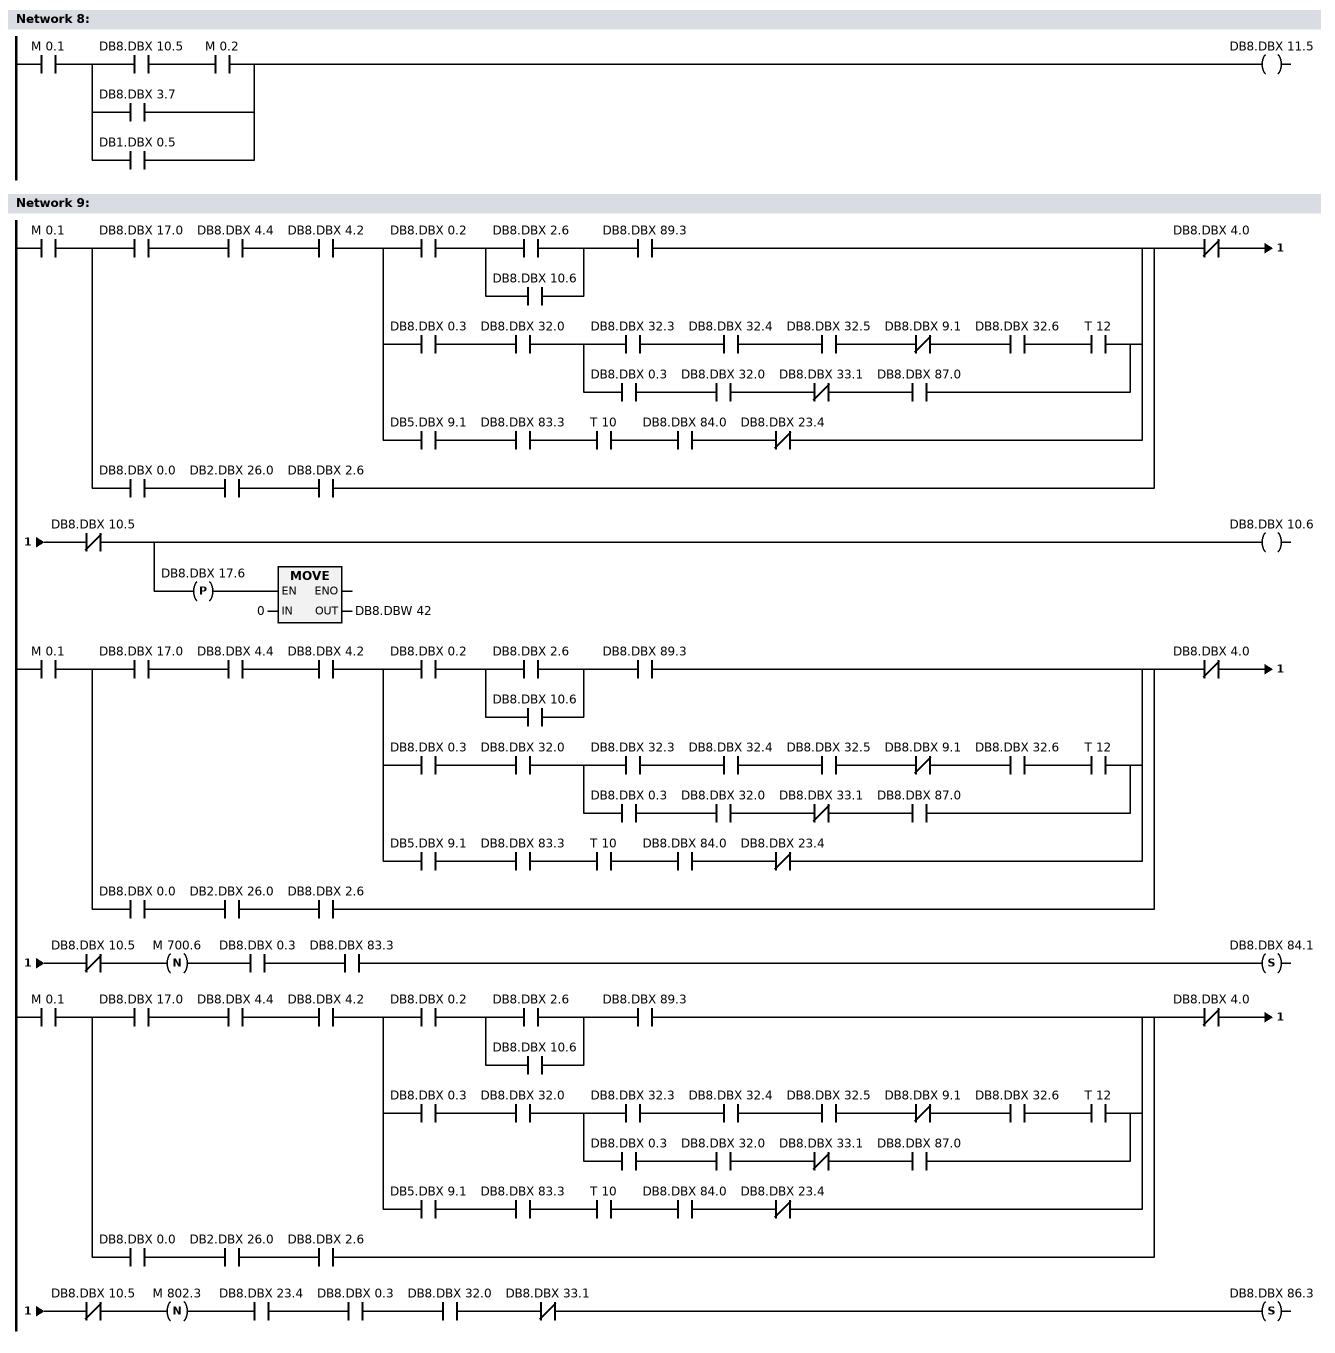
NETWORK
TITLE =
      A     M 0.1;
      A(;
      A     DB8.DBX 10.5;
      A     M 0.2;
      O     DB8.DBX 3.7;
      O     DB1.DBX 0.5;
      );
      =     DB8.DBX 11.5;
NETWORK
TITLE =
      A     M 0.1;
      A(;
      A     DB8.DBX 17.0;
      A     DB8.DBX 4.4;
      A     DB8.DBX 4.2;
      A(;
      A     DB8.DBX 0.2;
      A(;
      O     DB8.DBX 2.6;
      O     DB8.DBX 10.6;
      );
      A     DB8.DBX 89.3;
      O;
      A     DB8.DBX 0.3;
      A     DB8.DBX 32.0;
      A(;
      A     DB8.DBX 32.3;
      A     DB8.DBX 32.4;
      A     DB8.DBX 32.5;
      AN    DB8.DBX 9.1;
      A     DB8.DBX 32.6;
      A     T 12;
      O;
      A     DB8.DBX 0.3;
      A     DB8.DBX 32.0;
      AN    DB8.DBX 33.1;
      A     DB8.DBX 87.0;
      );
      O;
      A     DB5.DBX 9.1;
      A     DB8.DBX 83.3;
      A     T 10;
      A     DB8.DBX 84.0;
      AN    DB8.DBX 23.4;
      );
      O;
      A     DB8.DBX 0.0;
      A     DB2.DBX 26.0;
      A     DB8.DBX 2.6;
      );
      AN    DB8.DBX 4.0;
      AN    DB8.DBX 10.5;
      =     L 0.0;
      A     L 0.0;
      BLD   102;
      =     DB8.DBX 10.6;
      A     L 0.0;
      FP    DB8.DBX 17.6;
      JNB   M003;
      L     0;
      T     DB8.DBW 42;
M003: NOP   0;
      A(;
      A     L 0.0;
      FN    M 700.6;
      );
      A     DB8.DBX 0.3;
      A     DB8.DBX 83.3;
      S     DB8.DBX 84.1;
      A(;
      A     L 0.0;
      FN    M 802.3;
      );
      A     DB8.DBX 23.4;
      A     DB8.DBX 0.3;
      A     DB8.DBX 32.0;
      AN    DB8.DBX 33.1;
      S     DB8.DBX 86.3;
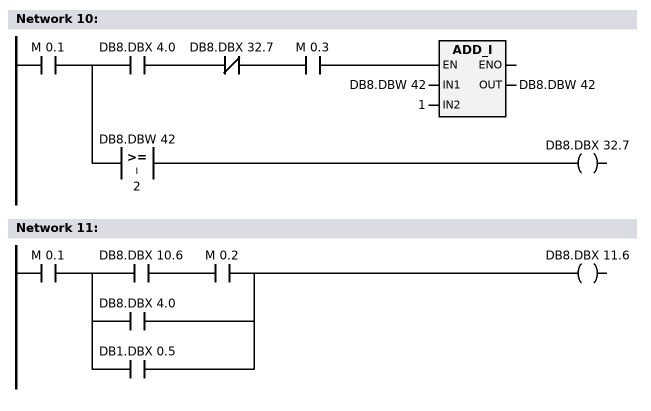
NETWORK
TITLE =
      A     M 0.1;
      =     L 0.0;
      A     L 0.0;
      A     DB8.DBX 4.0;
      AN    DB8.DBX 32.7;
      A     M 0.3;
      JNB   M004;
      L     DB8.DBW 42;
      L     1;
      +I;
      T     DB8.DBW 42;
M004: NOP   0;
      A     L 0.0;
      A(;
      L     DB8.DBW 42;
      L     2;
      >=I;
      );
      =     DB8.DBX 32.7;
NETWORK
TITLE =
      A     M 0.1;
      A(;
      A     DB8.DBX 10.6;
      A     M 0.2;
      O     DB8.DBX 4.0;
      O     DB1.DBX 0.5;
      );
      =     DB8.DBX 11.6;
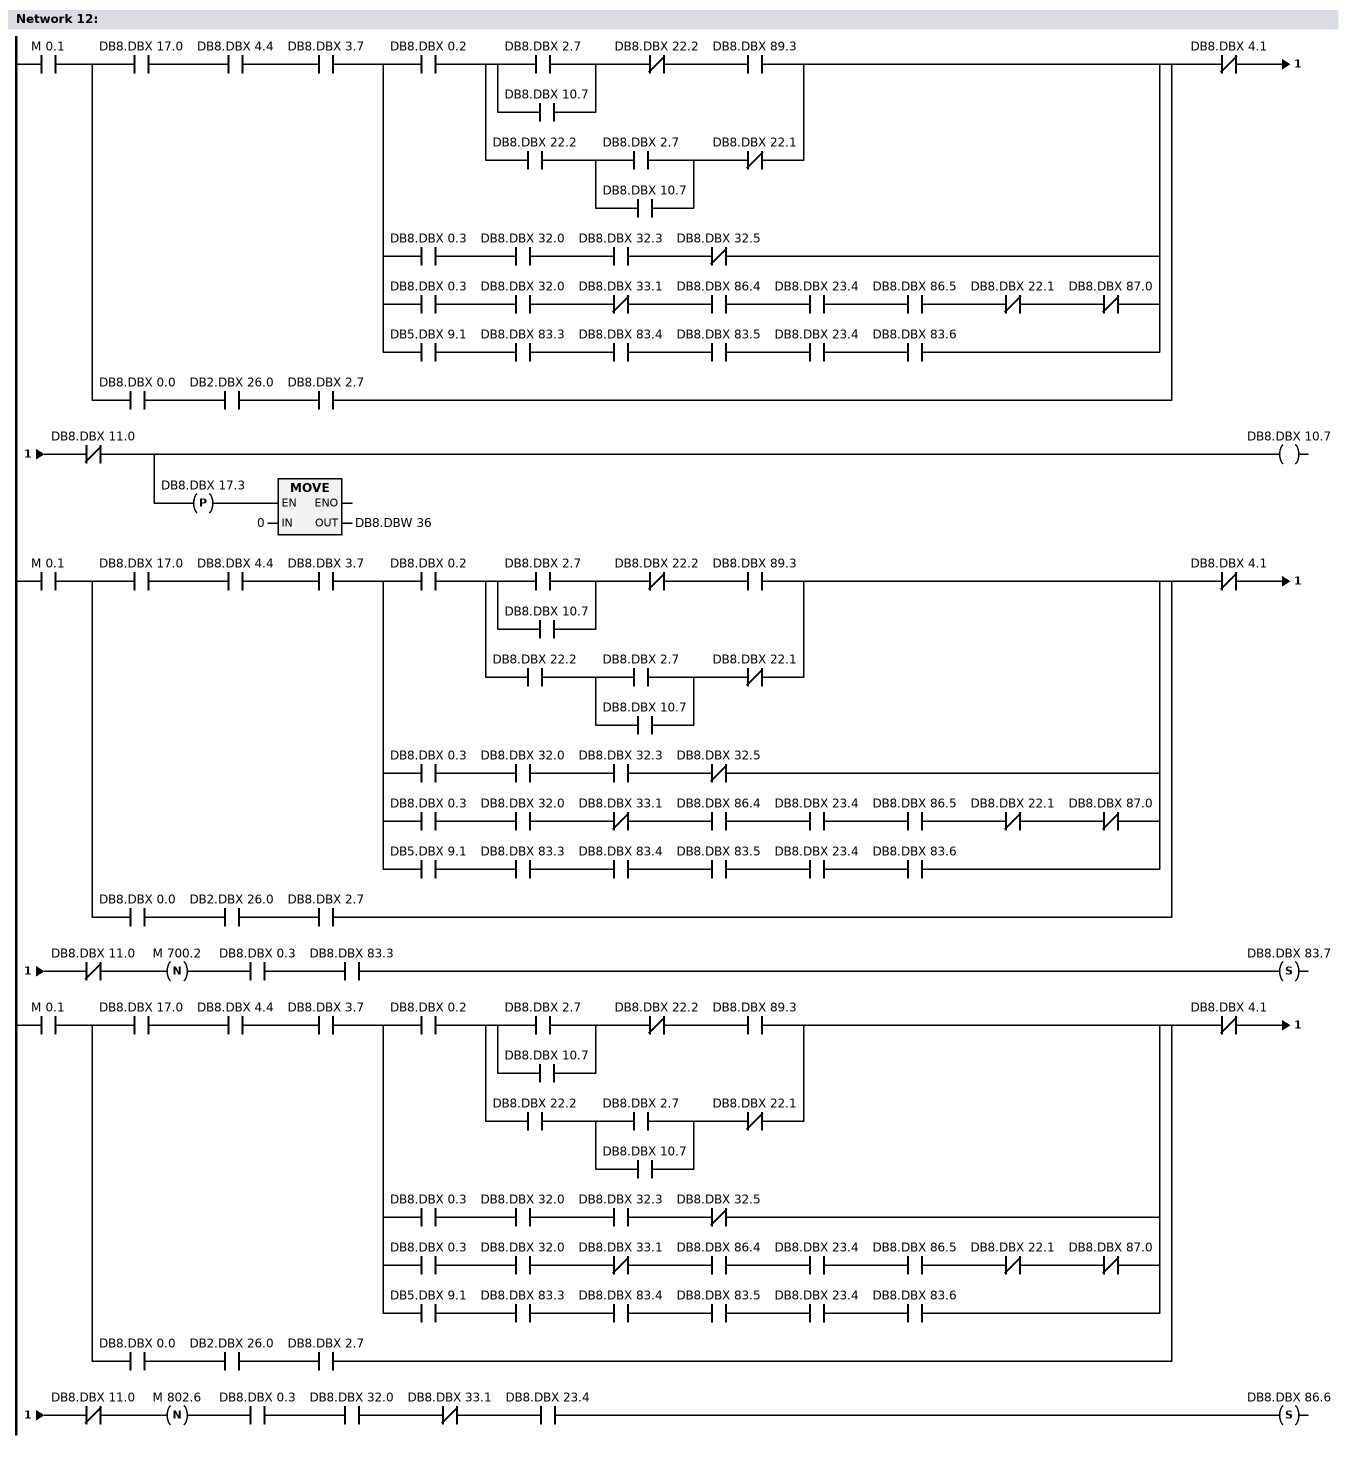
NETWORK
TITLE =
      A     M 0.1;
      A(;
      A     DB8.DBX 17.0;
      A     DB8.DBX 4.4;
      A     DB8.DBX 3.7;
      A(;
      A     DB8.DBX 0.2;
      A(;
      A(;
      O     DB8.DBX 2.7;
      O     DB8.DBX 10.7;
      );
      AN    DB8.DBX 22.2;
      A     DB8.DBX 89.3;
      O;
      A     DB8.DBX 22.2;
      A(;
      O     DB8.DBX 2.7;
      O     DB8.DBX 10.7;
      );
      AN    DB8.DBX 22.1;
      );
      O;
      A     DB8.DBX 0.3;
      A     DB8.DBX 32.0;
      A     DB8.DBX 32.3;
      AN    DB8.DBX 32.5;
      O;
      A     DB8.DBX 0.3;
      A     DB8.DBX 32.0;
      AN    DB8.DBX 33.1;
      A     DB8.DBX 86.4;
      A     DB8.DBX 23.4;
      A     DB8.DBX 86.5;
      AN    DB8.DBX 22.1;
      AN    DB8.DBX 87.0;
      O;
      A     DB5.DBX 9.1;
      A     DB8.DBX 83.3;
      A     DB8.DBX 83.4;
      A     DB8.DBX 83.5;
      A     DB8.DBX 23.4;
      A     DB8.DBX 83.6;
      );
      O;
      A     DB8.DBX 0.0;
      A     DB2.DBX 26.0;
      A     DB8.DBX 2.7;
      );
      AN    DB8.DBX 4.1;
      AN    DB8.DBX 11.0;
      =     L 0.0;
      A     L 0.0;
      BLD   102;
      =     DB8.DBX 10.7;
      A     L 0.0;
      FP    DB8.DBX 17.3;
      JNB   M005;
      L     0;
      T     DB8.DBW 36;
M005: NOP   0;
      A(;
      A     L 0.0;
      FN    M 700.2;
      );
      A     DB8.DBX 0.3;
      A     DB8.DBX 83.3;
      S     DB8.DBX 83.7;
      A(;
      A     L 0.0;
      FN    M 802.6;
      );
      A     DB8.DBX 0.3;
      A     DB8.DBX 32.0;
      AN    DB8.DBX 33.1;
      A     DB8.DBX 23.4;
      S     DB8.DBX 86.6;
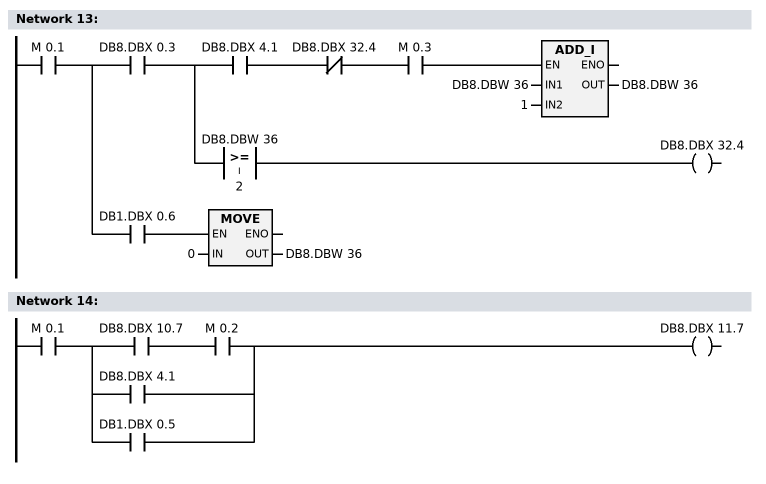
NETWORK
TITLE =
      A     M 0.1;
      =     L 0.0;
      A     L 0.0;
      A     DB8.DBX 0.3;
      =     L 0.1;
      A     L 0.1;
      A     DB8.DBX 4.1;
      AN    DB8.DBX 32.4;
      A     M 0.3;
      JNB   M006;
      L     DB8.DBW 36;
      L     1;
      +I;
      T     DB8.DBW 36;
M006: NOP   0;
      A     L 0.1;
      A(;
      L     DB8.DBW 36;
      L     2;
      >=I;
      );
      =     DB8.DBX 32.4;
      A     L 0.0;
      A     DB1.DBX 0.6;
      JNB   M007;
      L     0;
      T     DB8.DBW 36;
M007: NOP   0;
NETWORK
TITLE =
      A     M 0.1;
      A(;
      A     DB8.DBX 10.7;
      A     M 0.2;
      O     DB8.DBX 4.1;
      O     DB1.DBX 0.5;
      );
      =     DB8.DBX 11.7;
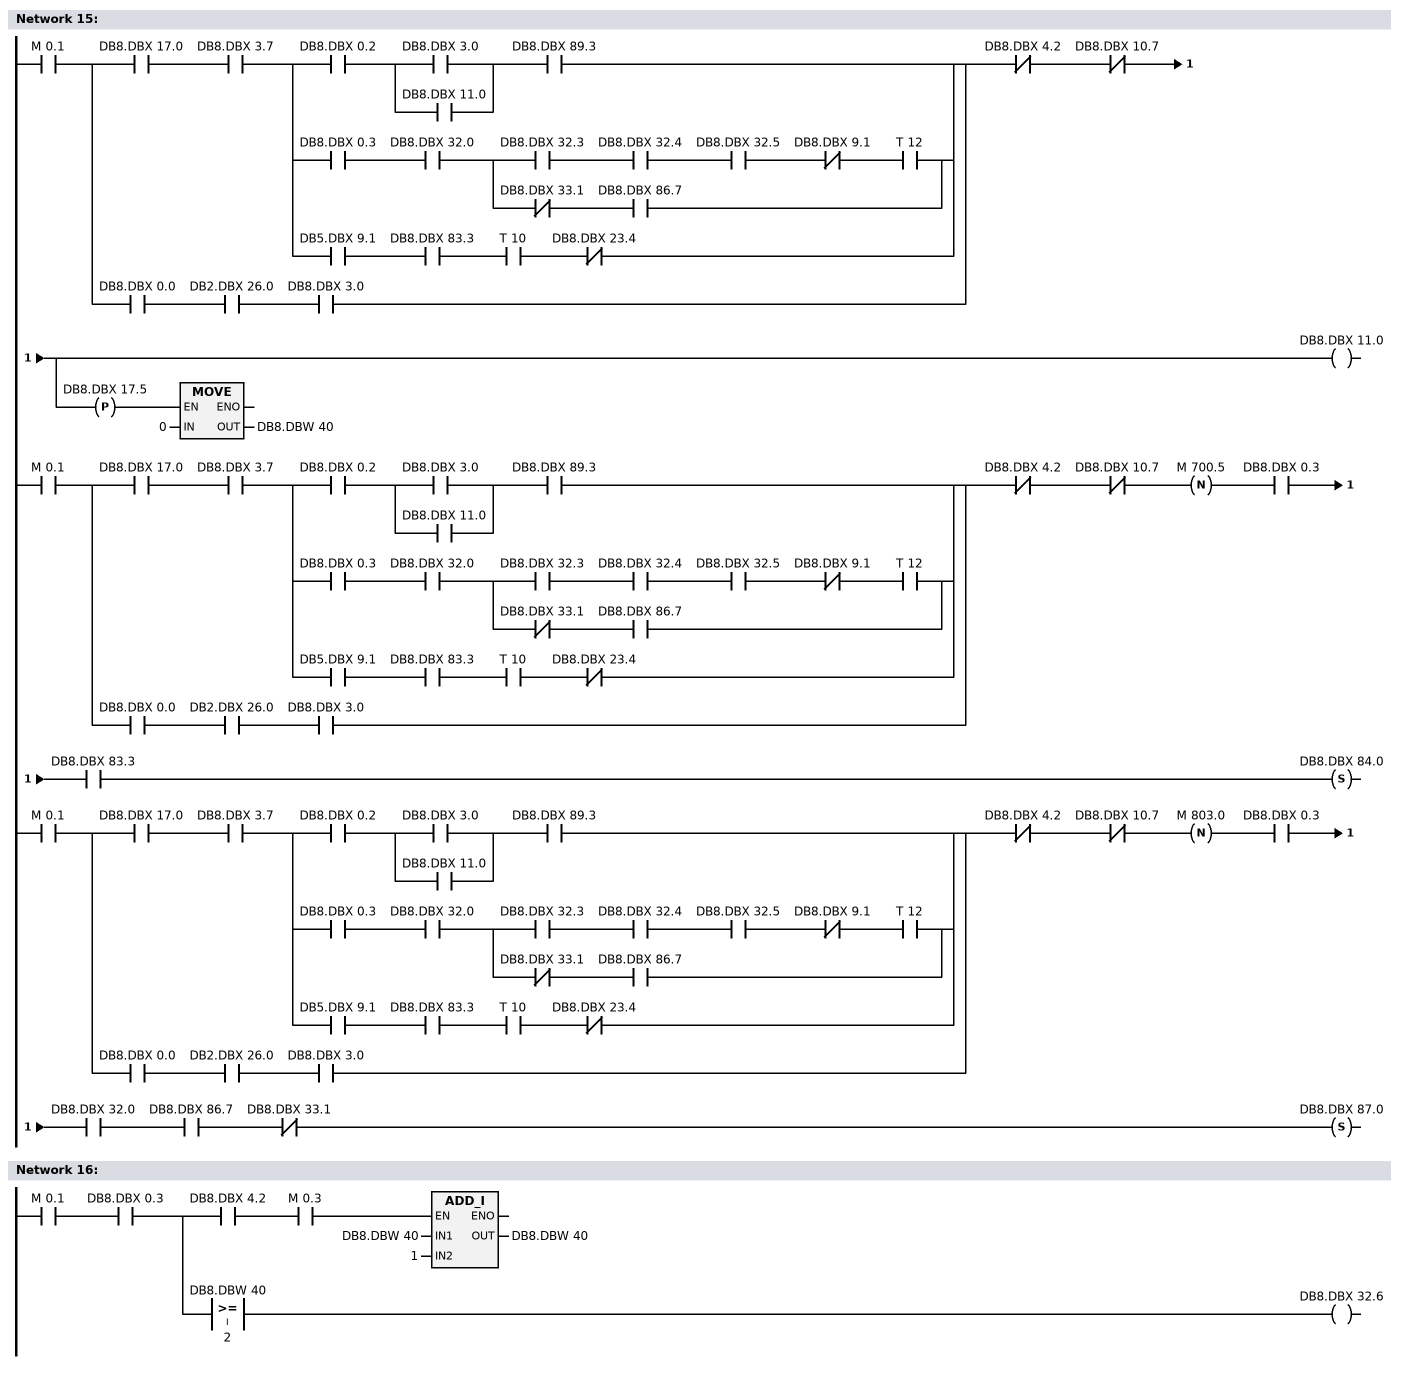
NETWORK
TITLE =
      A     M 0.1;
      A(;
      A     DB8.DBX 17.0;
      A     DB8.DBX 3.7;
      A(;
      A     DB8.DBX 0.2;
      A(;
      O     DB8.DBX 3.0;
      O     DB8.DBX 11.0;
      );
      A     DB8.DBX 89.3;
      O;
      A     DB8.DBX 0.3;
      A     DB8.DBX 32.0;
      A(;
      A     DB8.DBX 32.3;
      A     DB8.DBX 32.4;
      A     DB8.DBX 32.5;
      AN    DB8.DBX 9.1;
      A     T 12;
      O;
      AN    DB8.DBX 33.1;
      A     DB8.DBX 86.7;
      );
      O;
      A     DB5.DBX 9.1;
      A     DB8.DBX 83.3;
      A     T 10;
      AN    DB8.DBX 23.4;
      );
      O;
      A     DB8.DBX 0.0;
      A     DB2.DBX 26.0;
      A     DB8.DBX 3.0;
      );
      AN    DB8.DBX 4.2;
      AN    DB8.DBX 10.7;
      =     L 0.0;
      A     L 0.0;
      BLD   102;
      =     DB8.DBX 11.0;
      A     L 0.0;
      FP    DB8.DBX 17.5;
      JNB   M008;
      L     0;
      T     DB8.DBW 40;
M008: NOP   0;
      A(;
      A     L 0.0;
      FN    M 700.5;
      );
      A     DB8.DBX 0.3;
      A     DB8.DBX 83.3;
      S     DB8.DBX 84.0;
      A(;
      A     L 0.0;
      FN    M 803.0;
      );
      A     DB8.DBX 0.3;
      A     DB8.DBX 32.0;
      A     DB8.DBX 86.7;
      AN    DB8.DBX 33.1;
      S     DB8.DBX 87.0;
NETWORK
TITLE =
      A     M 0.1;
      A     DB8.DBX 0.3;
      =     L 0.0;
      A     L 0.0;
      A     DB8.DBX 4.2;
      A     M 0.3;
      JNB   M009;
      L     DB8.DBW 40;
      L     1;
      +I;
      T     DB8.DBW 40;
M009: NOP   0;
      A     L 0.0;
      A(;
      L     DB8.DBW 40;
      L     2;
      >=I;
      );
      =     DB8.DBX 32.6;
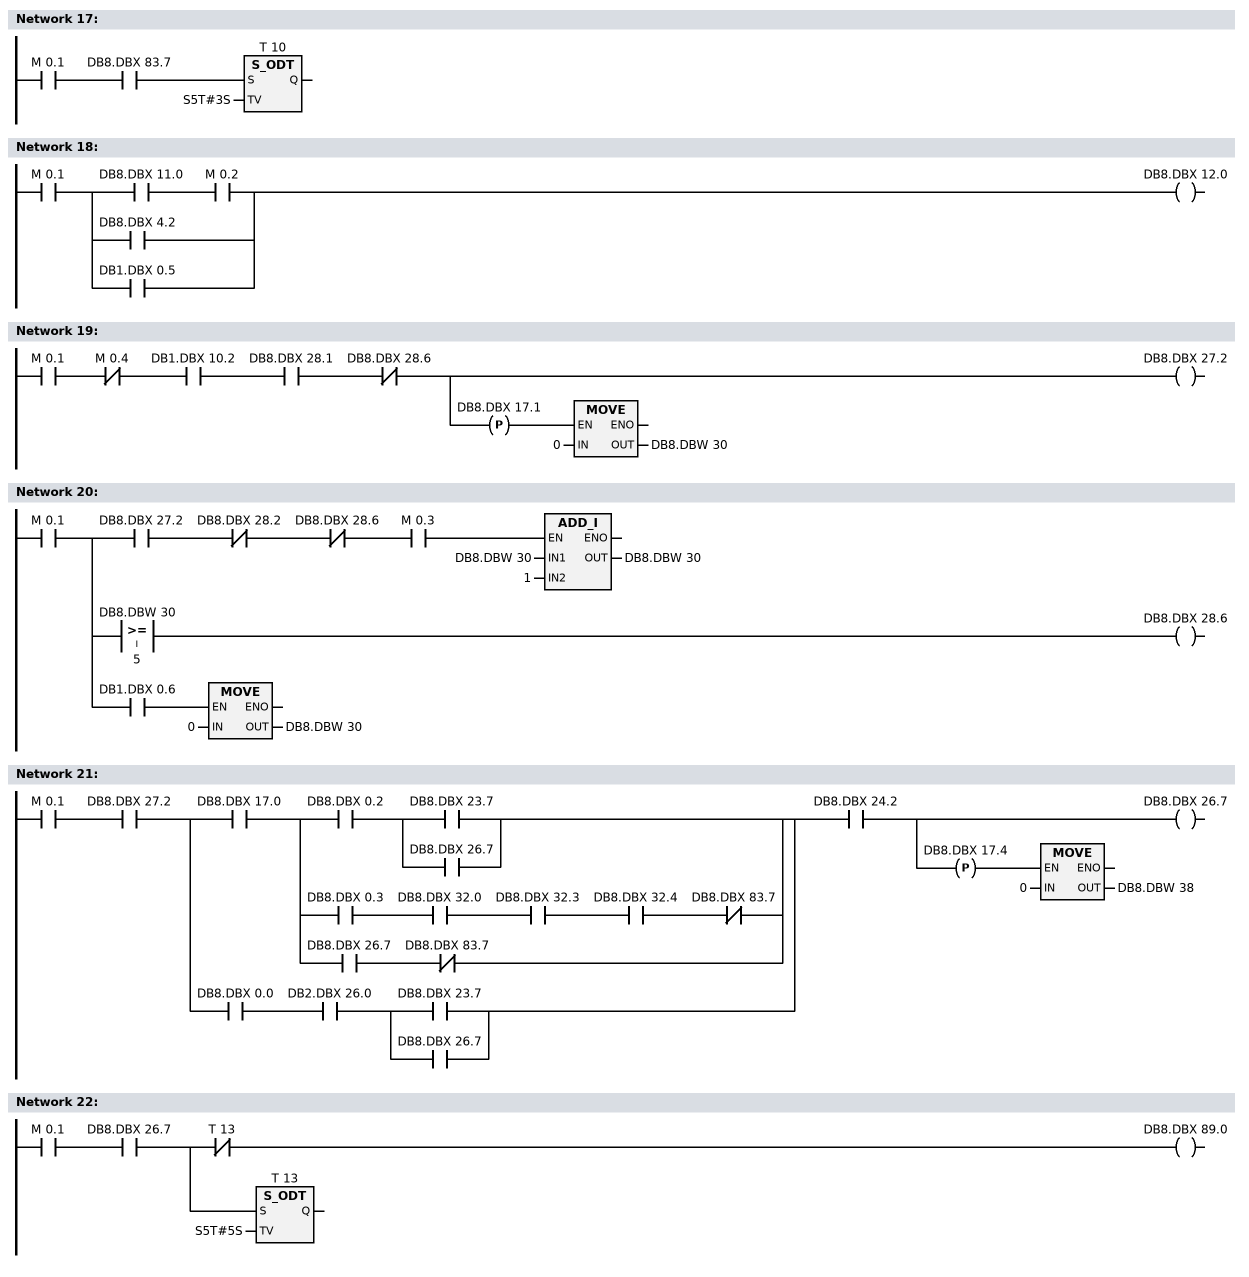
NETWORK
TITLE =
      A     M 0.1;
      A     DB8.DBX 83.7;
      L     S5T#3S;
      SD    T 10;
      NOP   0;
      NOP   0;
      NOP   0;
      NOP   0;
NETWORK
TITLE =
      A     M 0.1;
      A(;
      A     DB8.DBX 11.0;
      A     M 0.2;
      O     DB8.DBX 4.2;
      O     DB1.DBX 0.5;
      );
      =     DB8.DBX 12.0;
NETWORK
TITLE =
      A     M 0.1;
      AN    M 0.4;
      A     DB1.DBX 10.2;
      A     DB8.DBX 28.1;
      AN    DB8.DBX 28.6;
      =     L 0.0;
      A     L 0.0;
      BLD   102;
      =     DB8.DBX 27.2;
      A     L 0.0;
      FP    DB8.DBX 17.1;
      JNB   M010;
      L     0;
      T     DB8.DBW 30;
M010: NOP   0;
NETWORK
TITLE =
      A     M 0.1;
      =     L 0.0;
      A     L 0.0;
      A     DB8.DBX 27.2;
      AN    DB8.DBX 28.2;
      AN    DB8.DBX 28.6;
      A     M 0.3;
      JNB   M011;
      L     DB8.DBW 30;
      L     1;
      +I;
      T     DB8.DBW 30;
M011: NOP   0;
      A     L 0.0;
      A(;
      L     DB8.DBW 30;
      L     5;
      >=I;
      );
      =     DB8.DBX 28.6;
      A     L 0.0;
      A     DB1.DBX 0.6;
      JNB   M012;
      L     0;
      T     DB8.DBW 30;
M012: NOP   0;
NETWORK
TITLE =
      A     M 0.1;
      A     DB8.DBX 27.2;
      A(;
      A     DB8.DBX 17.0;
      A(;
      A     DB8.DBX 0.2;
      A(;
      O     DB8.DBX 23.7;
      O     DB8.DBX 26.7;
      );
      O;
      A     DB8.DBX 0.3;
      A     DB8.DBX 32.0;
      A     DB8.DBX 32.3;
      A     DB8.DBX 32.4;
      AN    DB8.DBX 83.7;
      O;
      A     DB8.DBX 26.7;
      AN    DB8.DBX 83.7;
      );
      O;
      A     DB8.DBX 0.0;
      A     DB2.DBX 26.0;
      A(;
      O     DB8.DBX 23.7;
      O     DB8.DBX 26.7;
      );
      );
      A     DB8.DBX 24.2;
      =     L 0.0;
      A     L 0.0;
      BLD   102;
      =     DB8.DBX 26.7;
      A     L 0.0;
      FP    DB8.DBX 17.4;
      JNB   M013;
      L     0;
      T     DB8.DBW 38;
M013: NOP   0;
NETWORK
TITLE =
      A     M 0.1;
      A     DB8.DBX 26.7;
      =     L 0.0;
      A     L 0.0;
      AN    T 13;
      =     DB8.DBX 89.0;
      A     L 0.0;
      L     S5T#5S;
      SD    T 13;
      NOP   0;
      NOP   0;
      NOP   0;
      NOP   0;
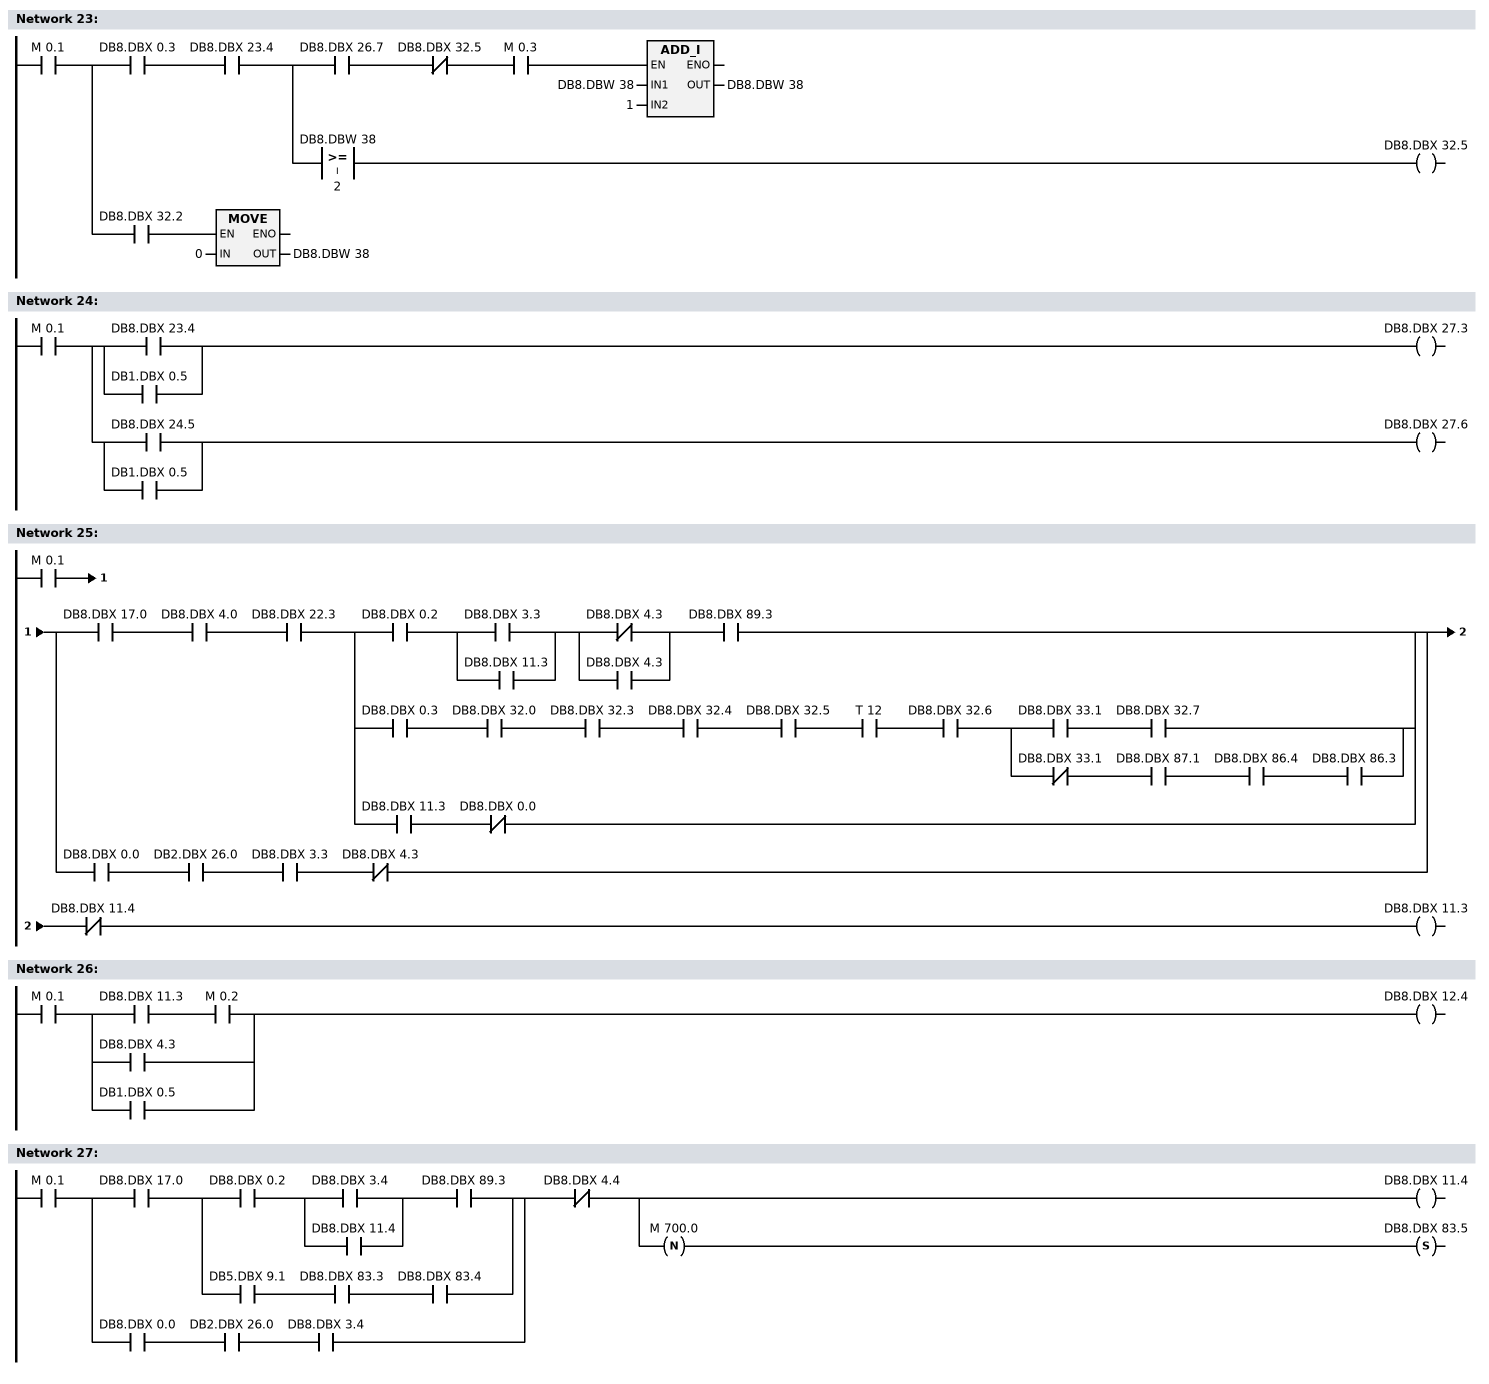
NETWORK
TITLE =
      A     M 0.1;
      =     L 0.0;
      A     L 0.0;
      A     DB8.DBX 0.3;
      A     DB8.DBX 23.4;
      =     L 0.1;
      A     L 0.1;
      A     DB8.DBX 26.7;
      AN    DB8.DBX 32.5;
      A     M 0.3;
      JNB   M014;
      L     DB8.DBW 38;
      L     1;
      +I;
      T     DB8.DBW 38;
M014: NOP   0;
      A     L 0.1;
      A(;
      L     DB8.DBW 38;
      L     2;
      >=I;
      );
      =     DB8.DBX 32.5;
      A     L 0.0;
      A     DB8.DBX 32.2;
      JNB   M015;
      L     0;
      T     DB8.DBW 38;
M015: NOP   0;
NETWORK
TITLE =
      A     M 0.1;
      =     L 0.0;
      A     L 0.0;
      A(;
      O     DB8.DBX 23.4;
      O     DB1.DBX 0.5;
      );
      =     DB8.DBX 27.3;
      A     L 0.0;
      A(;
      O     DB8.DBX 24.5;
      O     DB1.DBX 0.5;
      );
      =     DB8.DBX 27.6;
NETWORK
TITLE =
      A     M 0.1;
      A(;
      A     DB8.DBX 17.0;
      A     DB8.DBX 4.0;
      A     DB8.DBX 22.3;
      A(;
      A     DB8.DBX 0.2;
      A(;
      O     DB8.DBX 3.3;
      O     DB8.DBX 11.3;
      );
      A(;
      ON    DB8.DBX 4.3;
      O     DB8.DBX 4.3;
      );
      A     DB8.DBX 89.3;
      O;
      A     DB8.DBX 0.3;
      A     DB8.DBX 32.0;
      A     DB8.DBX 32.3;
      A     DB8.DBX 32.4;
      A     DB8.DBX 32.5;
      A     T 12;
      A     DB8.DBX 32.6;
      A(;
      A     DB8.DBX 33.1;
      A     DB8.DBX 32.7;
      O;
      AN    DB8.DBX 33.1;
      A     DB8.DBX 87.1;
      A     DB8.DBX 86.4;
      A     DB8.DBX 86.3;
      );
      O;
      A     DB8.DBX 11.3;
      AN    DB8.DBX 0.0;
      );
      O;
      A     DB8.DBX 0.0;
      A     DB2.DBX 26.0;
      A     DB8.DBX 3.3;
      AN    DB8.DBX 4.3;
      );
      AN    DB8.DBX 11.4;
      =     DB8.DBX 11.3;
NETWORK
TITLE =
      A     M 0.1;
      A(;
      A     DB8.DBX 11.3;
      A     M 0.2;
      O     DB8.DBX 4.3;
      O     DB1.DBX 0.5;
      );
      =     DB8.DBX 12.4;
NETWORK
TITLE =
      A     M 0.1;
      A(;
      A     DB8.DBX 17.0;
      A(;
      A     DB8.DBX 0.2;
      A(;
      O     DB8.DBX 3.4;
      O     DB8.DBX 11.4;
      );
      A     DB8.DBX 89.3;
      O;
      A     DB5.DBX 9.1;
      A     DB8.DBX 83.3;
      A     DB8.DBX 83.4;
      );
      O;
      A     DB8.DBX 0.0;
      A     DB2.DBX 26.0;
      A     DB8.DBX 3.4;
      );
      AN    DB8.DBX 4.4;
      =     L 0.0;
      A     L 0.0;
      BLD   102;
      =     DB8.DBX 11.4;
      A     L 0.0;
      FN    M 700.0;
      S     DB8.DBX 83.5;
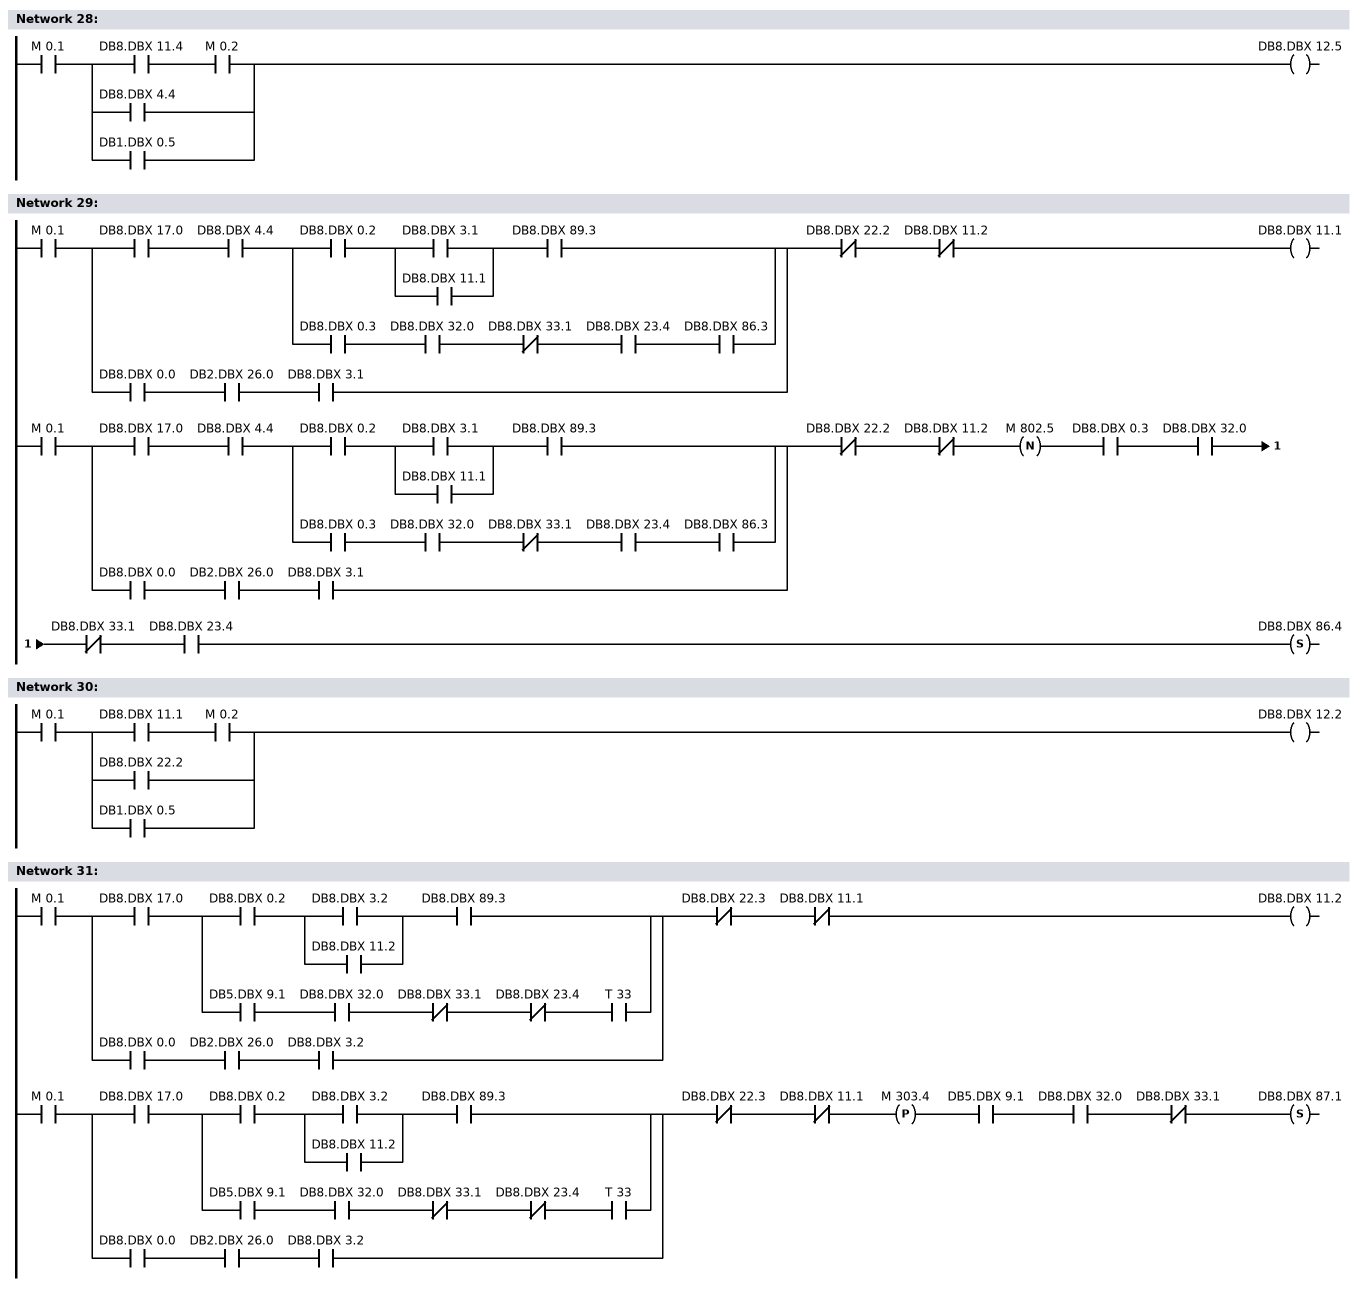
NETWORK
TITLE =
      A     M 0.1;
      A(;
      A     DB8.DBX 11.4;
      A     M 0.2;
      O     DB8.DBX 4.4;
      O     DB1.DBX 0.5;
      );
      =     DB8.DBX 12.5;
NETWORK
TITLE =
      A     M 0.1;
      A(;
      A     DB8.DBX 17.0;
      A     DB8.DBX 4.4;
      A(;
      A     DB8.DBX 0.2;
      A(;
      O     DB8.DBX 3.1;
      O     DB8.DBX 11.1;
      );
      A     DB8.DBX 89.3;
      O;
      A     DB8.DBX 0.3;
      A     DB8.DBX 32.0;
      AN    DB8.DBX 33.1;
      A     DB8.DBX 23.4;
      A     DB8.DBX 86.3;
      );
      O;
      A     DB8.DBX 0.0;
      A     DB2.DBX 26.0;
      A     DB8.DBX 3.1;
      );
      AN    DB8.DBX 22.2;
      AN    DB8.DBX 11.2;
      =     L 0.0;
      A     L 0.0;
      BLD   102;
      =     DB8.DBX 11.1;
      A(;
      A     L 0.0;
      FN    M 802.5;
      );
      A     DB8.DBX 0.3;
      A     DB8.DBX 32.0;
      AN    DB8.DBX 33.1;
      A     DB8.DBX 23.4;
      S     DB8.DBX 86.4;
NETWORK
TITLE =
      A     M 0.1;
      A(;
      A     DB8.DBX 11.1;
      A     M 0.2;
      O     DB8.DBX 22.2;
      O     DB1.DBX 0.5;
      );
      =     DB8.DBX 12.2;
NETWORK
TITLE =
      A     M 0.1;
      A(;
      A     DB8.DBX 17.0;
      A(;
      A     DB8.DBX 0.2;
      A(;
      O     DB8.DBX 3.2;
      O     DB8.DBX 11.2;
      );
      A     DB8.DBX 89.3;
      O;
      A     DB5.DBX 9.1;
      A     DB8.DBX 32.0;
      AN    DB8.DBX 33.1;
      AN    DB8.DBX 23.4;
      A     T 33;
      );
      O;
      A     DB8.DBX 0.0;
      A     DB2.DBX 26.0;
      A     DB8.DBX 3.2;
      );
      AN    DB8.DBX 22.3;
      AN    DB8.DBX 11.1;
      =     L 0.0;
      A     L 0.0;
      BLD   102;
      =     DB8.DBX 11.2;
      A(;
      A     L 0.0;
      FP    M 303.4;
      );
      A     DB5.DBX 9.1;
      A     DB8.DBX 32.0;
      AN    DB8.DBX 33.1;
      S     DB8.DBX 87.1;
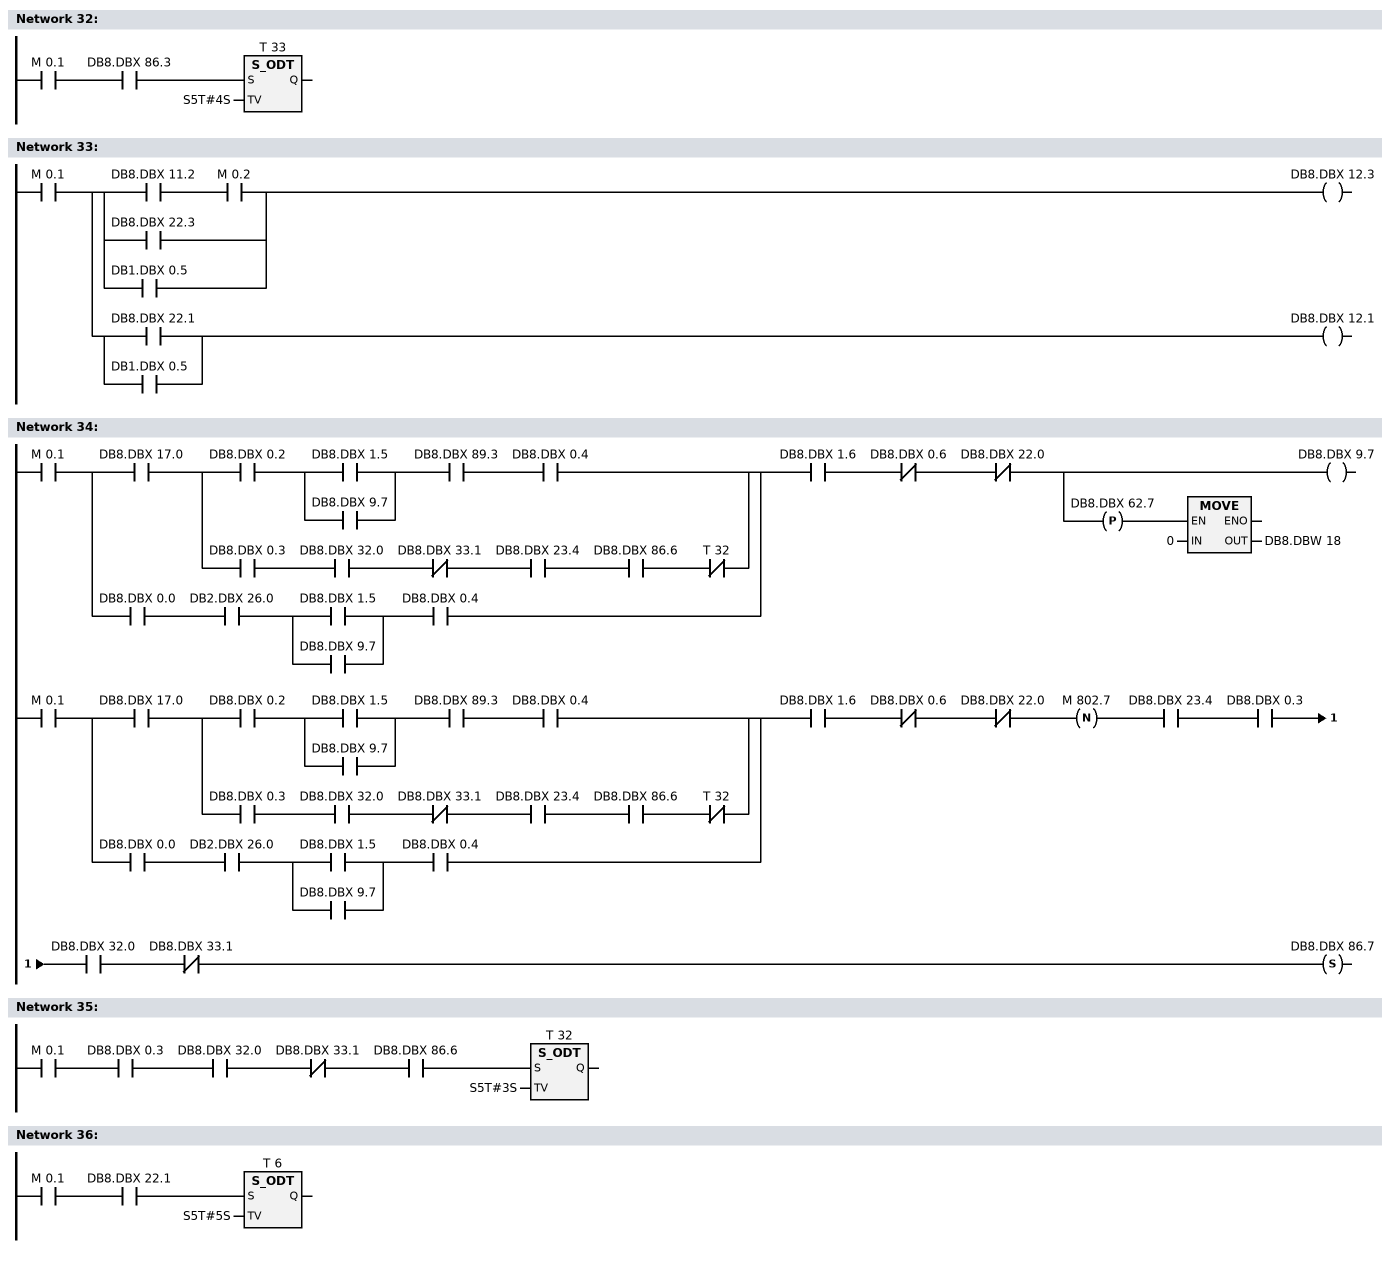
NETWORK
TITLE =
      A     M 0.1;
      A     DB8.DBX 86.3;
      L     S5T#4S;
      SD    T 33;
      NOP   0;
      NOP   0;
      NOP   0;
      NOP   0;
NETWORK
TITLE =
      A     M 0.1;
      =     L 0.0;
      A     L 0.0;
      A(;
      A     DB8.DBX 11.2;
      A     M 0.2;
      O     DB8.DBX 22.3;
      O     DB1.DBX 0.5;
      );
      =     DB8.DBX 12.3;
      A     L 0.0;
      A(;
      O     DB8.DBX 22.1;
      O     DB1.DBX 0.5;
      );
      =     DB8.DBX 12.1;
NETWORK
TITLE =
      A     M 0.1;
      A(;
      A     DB8.DBX 17.0;
      A(;
      A     DB8.DBX 0.2;
      A(;
      O     DB8.DBX 1.5;
      O     DB8.DBX 9.7;
      );
      A     DB8.DBX 89.3;
      A     DB8.DBX 0.4;
      O;
      A     DB8.DBX 0.3;
      A     DB8.DBX 32.0;
      AN    DB8.DBX 33.1;
      A     DB8.DBX 23.4;
      A     DB8.DBX 86.6;
      AN    T 32;
      );
      O;
      A     DB8.DBX 0.0;
      A     DB2.DBX 26.0;
      A(;
      O     DB8.DBX 1.5;
      O     DB8.DBX 9.7;
      );
      A     DB8.DBX 0.4;
      );
      A     DB8.DBX 1.6;
      AN    DB8.DBX 0.6;
      AN    DB8.DBX 22.0;
      =     L 0.0;
      A     L 0.0;
      BLD   102;
      =     DB8.DBX 9.7;
      A     L 0.0;
      FP    DB8.DBX 62.7;
      JNB   M016;
      L     0;
      T     DB8.DBW 18;
M016: NOP   0;
      A(;
      A     L 0.0;
      FN    M 802.7;
      );
      A     DB8.DBX 23.4;
      A     DB8.DBX 0.3;
      A     DB8.DBX 32.0;
      AN    DB8.DBX 33.1;
      S     DB8.DBX 86.7;
NETWORK
TITLE =
      A     M 0.1;
      A     DB8.DBX 0.3;
      A     DB8.DBX 32.0;
      AN    DB8.DBX 33.1;
      A     DB8.DBX 86.6;
      L     S5T#3S;
      SD    T 32;
      NOP   0;
      NOP   0;
      NOP   0;
      NOP   0;
NETWORK
TITLE =
      A     M 0.1;
      A     DB8.DBX 22.1;
      L     S5T#5S;
      SD    T 6;
      NOP   0;
      NOP   0;
      NOP   0;
      NOP   0;
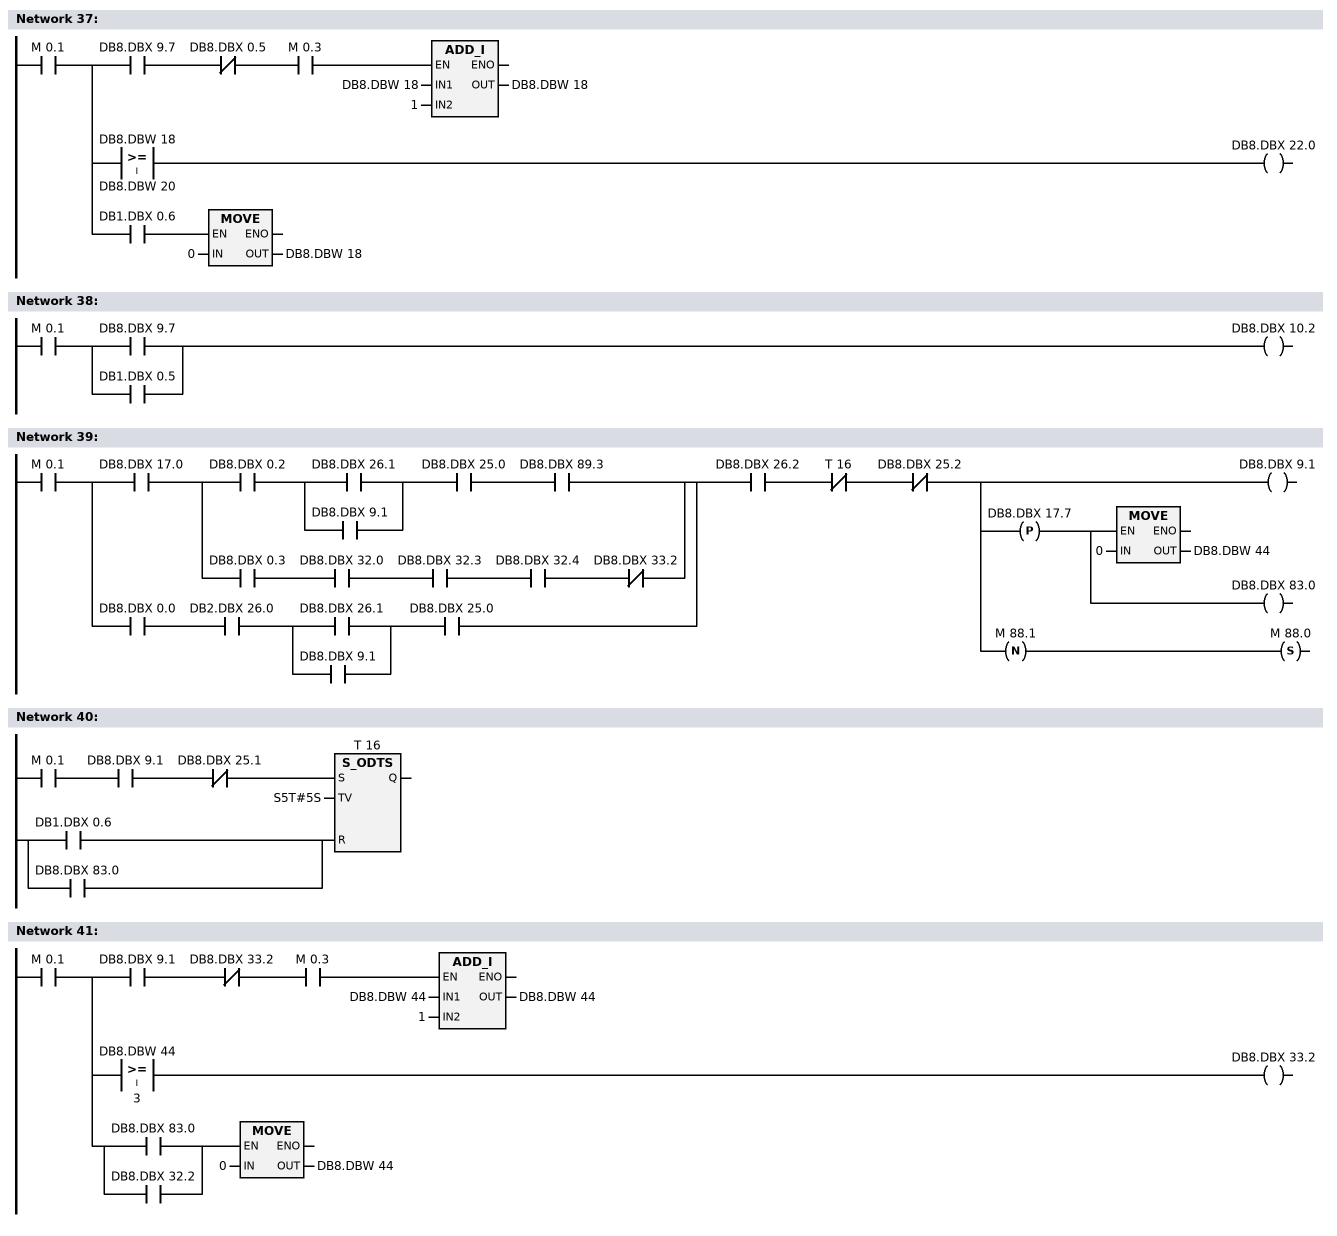
NETWORK
TITLE =
      A     M 0.1;
      =     L 0.0;
      A     L 0.0;
      A     DB8.DBX 9.7;
      AN    DB8.DBX 0.5;
      A     M 0.3;
      JNB   M017;
      L     DB8.DBW 18;
      L     1;
      +I;
      T     DB8.DBW 18;
M017: NOP   0;
      A     L 0.0;
      A(;
      L     DB8.DBW 18;
      L     DB8.DBW 20;
      >=I;
      );
      =     DB8.DBX 22.0;
      A     L 0.0;
      A     DB1.DBX 0.6;
      JNB   M018;
      L     0;
      T     DB8.DBW 18;
M018: NOP   0;
NETWORK
TITLE =
      A     M 0.1;
      A(;
      O     DB8.DBX 9.7;
      O     DB1.DBX 0.5;
      );
      =     DB8.DBX 10.2;
NETWORK
TITLE =
      A     M 0.1;
      A(;
      A     DB8.DBX 17.0;
      A(;
      A     DB8.DBX 0.2;
      A(;
      O     DB8.DBX 26.1;
      O     DB8.DBX 9.1;
      );
      A     DB8.DBX 25.0;
      A     DB8.DBX 89.3;
      O;
      A     DB8.DBX 0.3;
      A     DB8.DBX 32.0;
      A     DB8.DBX 32.3;
      A     DB8.DBX 32.4;
      AN    DB8.DBX 33.2;
      );
      O;
      A     DB8.DBX 0.0;
      A     DB2.DBX 26.0;
      A(;
      O     DB8.DBX 26.1;
      O     DB8.DBX 9.1;
      );
      A     DB8.DBX 25.0;
      );
      A     DB8.DBX 26.2;
      AN    T 16;
      AN    DB8.DBX 25.2;
      =     L 0.0;
      A     L 0.0;
      BLD   102;
      =     DB8.DBX 9.1;
      A     L 0.0;
      FP    DB8.DBX 17.7;
      =     L 0.1;
      A     L 0.1;
      JNB   M019;
      L     0;
      T     DB8.DBW 44;
M019: NOP   0;
      A     L 0.1;
      BLD   102;
      =     DB8.DBX 83.0;
      A     L 0.0;
      FN    M 88.1;
      S     M 88.0;
NETWORK
TITLE =
      A     M 0.1;
      A     DB8.DBX 9.1;
      AN    DB8.DBX 25.1;
      L     S5T#5S;
      SS    T 16;
      A(;
      O     DB1.DBX 0.6;
      O     DB8.DBX 83.0;
      );
      R     T 16;
      NOP   0;
      NOP   0;
      NOP   0;
NETWORK
TITLE =
      A     M 0.1;
      =     L 0.0;
      A     L 0.0;
      A     DB8.DBX 9.1;
      AN    DB8.DBX 33.2;
      A     M 0.3;
      JNB   M020;
      L     DB8.DBW 44;
      L     1;
      +I;
      T     DB8.DBW 44;
M020: NOP   0;
      A     L 0.0;
      A(;
      L     DB8.DBW 44;
      L     3;
      >=I;
      );
      =     DB8.DBX 33.2;
      A     L 0.0;
      A(;
      O     DB8.DBX 83.0;
      O     DB8.DBX 32.2;
      );
      JNB   M021;
      L     0;
      T     DB8.DBW 44;
M021: NOP   0;
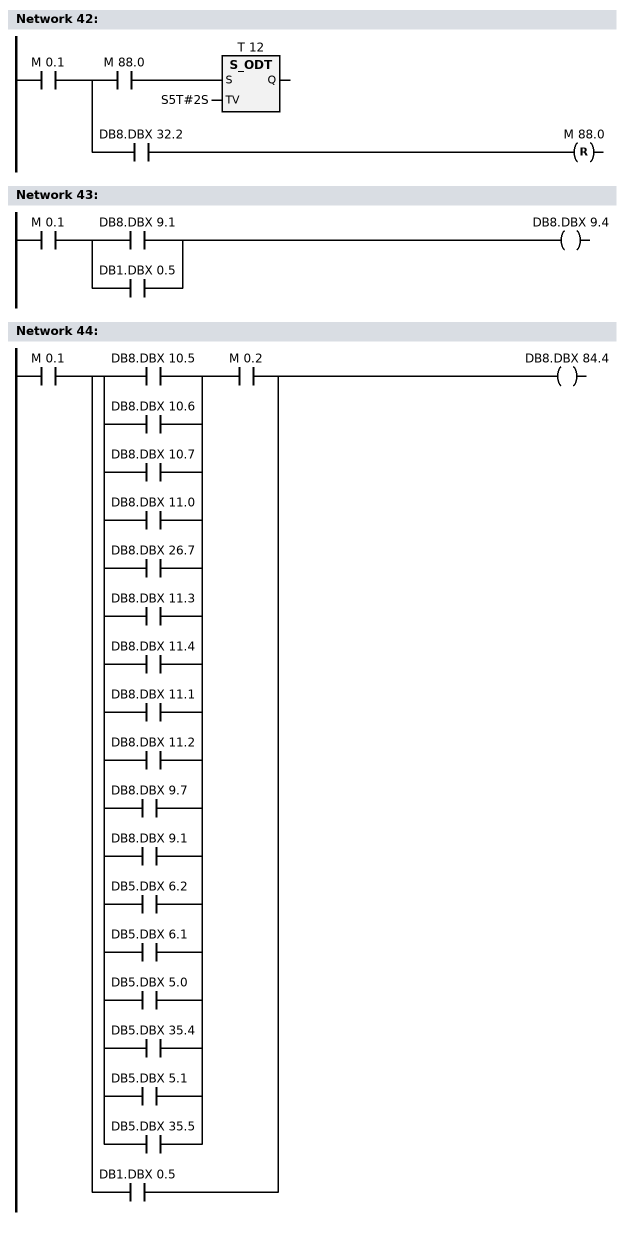
NETWORK
TITLE =
      A     M 0.1;
      =     L 0.0;
      A     L 0.0;
      A     M 88.0;
      L     S5T#2S;
      SD    T 12;
      NOP   0;
      NOP   0;
      NOP   0;
      NOP   0;
      A     L 0.0;
      A     DB8.DBX 32.2;
      R     M 88.0;
NETWORK
TITLE =
      A     M 0.1;
      A(;
      O     DB8.DBX 9.1;
      O     DB1.DBX 0.5;
      );
      =     DB8.DBX 9.4;
NETWORK
TITLE =
      A     M 0.1;
      A(;
      A(;
      O     DB8.DBX 10.5;
      O     DB8.DBX 10.6;
      O     DB8.DBX 10.7;
      O     DB8.DBX 11.0;
      O     DB8.DBX 26.7;
      O     DB8.DBX 11.3;
      O     DB8.DBX 11.4;
      O     DB8.DBX 11.1;
      O     DB8.DBX 11.2;
      O     DB8.DBX 9.7;
      O     DB8.DBX 9.1;
      O     DB5.DBX 6.2;
      O     DB5.DBX 6.1;
      O     DB5.DBX 5.0;
      O     DB5.DBX 35.4;
      O     DB5.DBX 5.1;
      O     DB5.DBX 35.5;
      );
      A     M 0.2;
      O     DB1.DBX 0.5;
      );
      =     DB8.DBX 84.4;
END_FUNCTION

FUNCTION FC 12 : VOID
AUTHOR : Arun_Ram
VERSION : 0.1
BEGIN
// (block stored without names or comments; labels and parameter names are numbered)
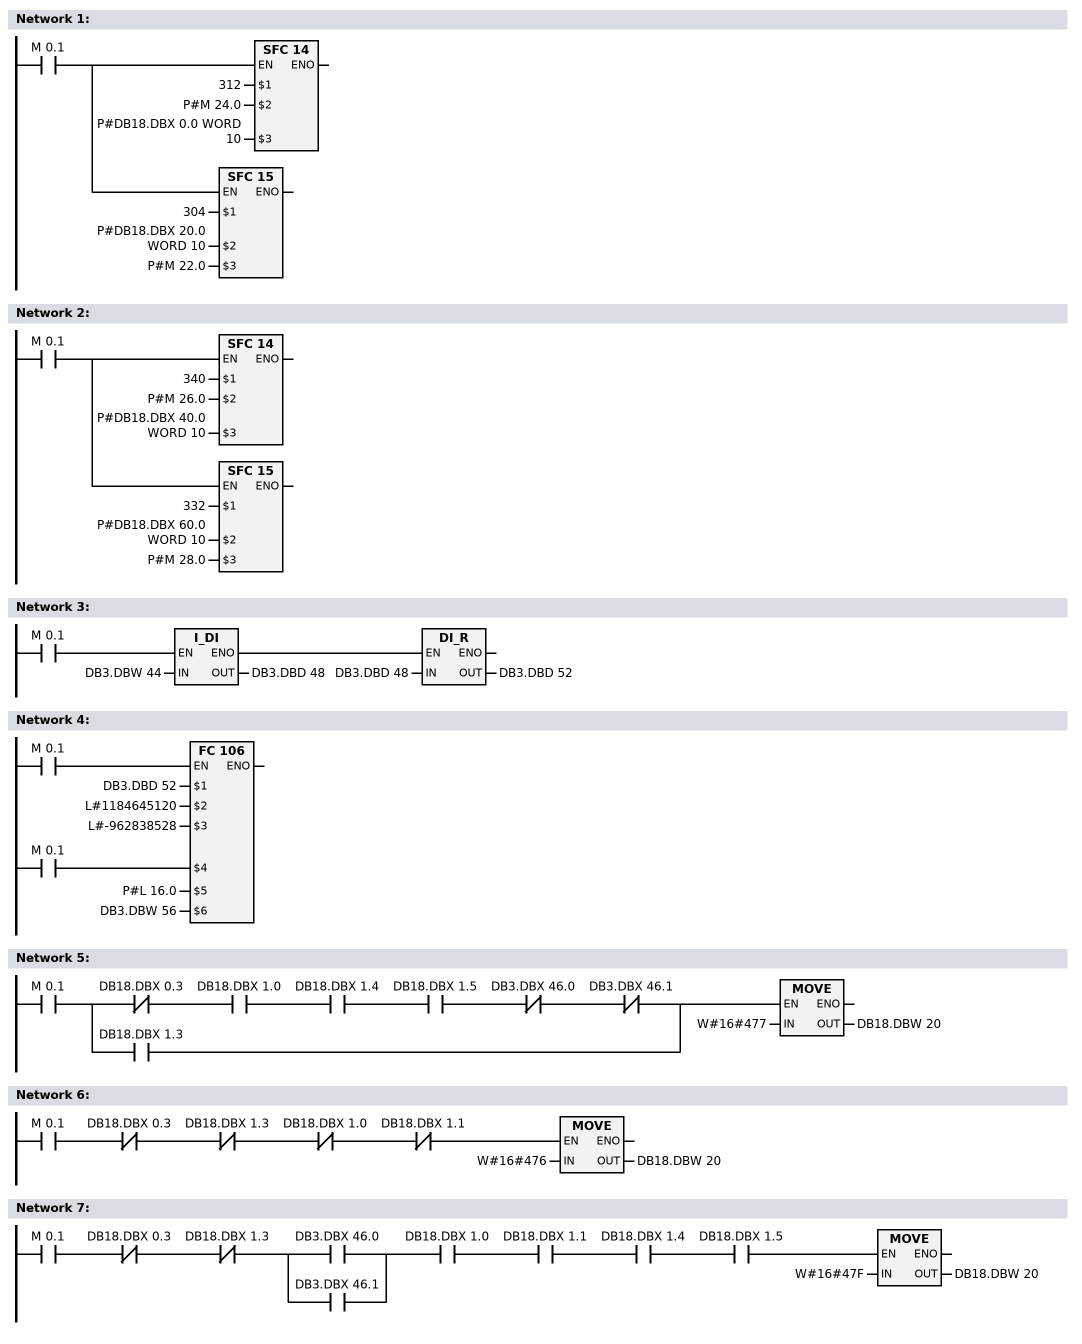
NETWORK
TITLE =
      A     M 0.1;
      =     L 36.0;
      A     L 36.0;
      JNB   M001;
      CALL  SFC 14 (
           $1                       := 312,
           $2                       := P#M 24.0,
           $3                       := P#DB18.DBX 0.0 WORD 10);
M001: NOP   0;
      A     L 36.0;
      JNB   M002;
      CALL  SFC 15 (
           $1                       := 304,
           $2                       := P#DB18.DBX 20.0 WORD 10,
           $3                       := P#M 22.0);
M002: NOP   0;
NETWORK
TITLE =
      A     M 0.1;
      =     L 36.0;
      A     L 36.0;
      JNB   M003;
      CALL  SFC 14 (
           $1                       := 340,
           $2                       := P#M 26.0,
           $3                       := P#DB18.DBX 40.0 WORD 10);
M003: NOP   0;
      A     L 36.0;
      JNB   M004;
      CALL  SFC 15 (
           $1                       := 332,
           $2                       := P#DB18.DBX 60.0 WORD 10,
           $3                       := P#M 28.0);
M004: NOP   0;
NETWORK
TITLE =
      A(;
      A     M 0.1;
      JNB   M005;
      L     DB3.DBW 44;
      ITD;
      T     DB3.DBD 48;
      SET;
      SAVE;
      CLR;
M005: A     BR;
      );
      JNB   M006;
      L     DB3.DBD 48;
      DTR;
      T     DB3.DBD 52;
M006: NOP   0;
NETWORK
TITLE =
      A     M 0.1;
      =     L 36.0;
      BLD   103;
      A     M 0.1;
      JNB   M007;
      CALL  FC 106 (
           $1                       := DB3.DBD 52,
           $2                       := L#1184645120,
           $3                       := L#-962838528,
           $4                       := L 36.0,
           $5                       := P#L 16.0,
           $6                       := DB3.DBW 56);
M007: NOP   0;
NETWORK
TITLE =
      A     M 0.1;
      A(;
      AN    DB18.DBX 0.3;
      A     DB18.DBX 1.0;
      A     DB18.DBX 1.4;
      A     DB18.DBX 1.5;
      AN    DB3.DBX 46.0;
      AN    DB3.DBX 46.1;
      O     DB18.DBX 1.3;
      );
      JNB   M008;
      L     W#16#477;
      T     DB18.DBW 20;
M008: NOP   0;
NETWORK
TITLE =
      A     M 0.1;
      AN    DB18.DBX 0.3;
      AN    DB18.DBX 1.3;
      AN    DB18.DBX 1.0;
      AN    DB18.DBX 1.1;
      JNB   M009;
      L     W#16#476;
      T     DB18.DBW 20;
M009: NOP   0;
NETWORK
TITLE =
      A     M 0.1;
      AN    DB18.DBX 0.3;
      AN    DB18.DBX 1.3;
      A(;
      O     DB3.DBX 46.0;
      O     DB3.DBX 46.1;
      );
      A     DB18.DBX 1.0;
      A     DB18.DBX 1.1;
      A     DB18.DBX 1.4;
      A     DB18.DBX 1.5;
      JNB   M010;
      L     W#16#47F;
      T     DB18.DBW 20;
M010: NOP   0;
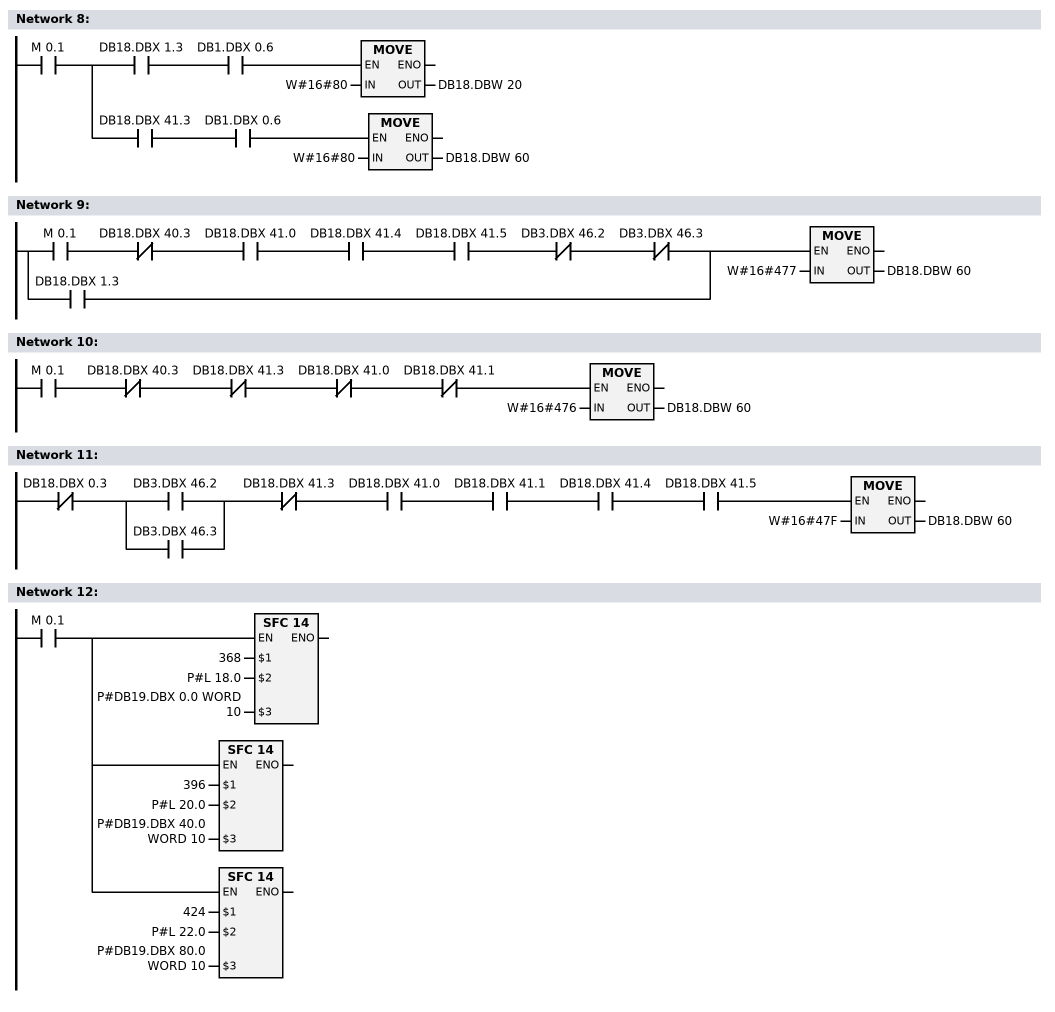
NETWORK
TITLE =
      A     M 0.1;
      =     L 36.0;
      A     L 36.0;
      A     DB18.DBX 1.3;
      A     DB1.DBX 0.6;
      JNB   M011;
      L     W#16#80;
      T     DB18.DBW 20;
M011: NOP   0;
      A     L 36.0;
      A     DB18.DBX 41.3;
      A     DB1.DBX 0.6;
      JNB   M012;
      L     W#16#80;
      T     DB18.DBW 60;
M012: NOP   0;
NETWORK
TITLE =
      A(;
      A     M 0.1;
      AN    DB18.DBX 40.3;
      A     DB18.DBX 41.0;
      A     DB18.DBX 41.4;
      A     DB18.DBX 41.5;
      AN    DB3.DBX 46.2;
      AN    DB3.DBX 46.3;
      O     DB18.DBX 1.3;
      );
      JNB   M013;
      L     W#16#477;
      T     DB18.DBW 60;
M013: NOP   0;
NETWORK
TITLE =
      A     M 0.1;
      AN    DB18.DBX 40.3;
      AN    DB18.DBX 41.3;
      AN    DB18.DBX 41.0;
      AN    DB18.DBX 41.1;
      JNB   M014;
      L     W#16#476;
      T     DB18.DBW 60;
M014: NOP   0;
NETWORK
TITLE =
      AN    DB18.DBX 0.3;
      A(;
      O     DB3.DBX 46.2;
      O     DB3.DBX 46.3;
      );
      AN    DB18.DBX 41.3;
      A     DB18.DBX 41.0;
      A     DB18.DBX 41.1;
      A     DB18.DBX 41.4;
      A     DB18.DBX 41.5;
      JNB   M015;
      L     W#16#47F;
      T     DB18.DBW 60;
M015: NOP   0;
NETWORK
TITLE =
      A     M 0.1;
      =     L 36.0;
      A     L 36.0;
      JNB   M016;
      CALL  SFC 14 (
           $1                       := 368,
           $2                       := P#L 18.0,
           $3                       := P#DB19.DBX 0.0 WORD 10);
M016: NOP   0;
      A     L 36.0;
      JNB   M017;
      CALL  SFC 14 (
           $1                       := 396,
           $2                       := P#L 20.0,
           $3                       := P#DB19.DBX 40.0 WORD 10);
M017: NOP   0;
      A     L 36.0;
      JNB   M018;
      CALL  SFC 14 (
           $1                       := 424,
           $2                       := P#L 22.0,
           $3                       := P#DB19.DBX 80.0 WORD 10);
M018: NOP   0;
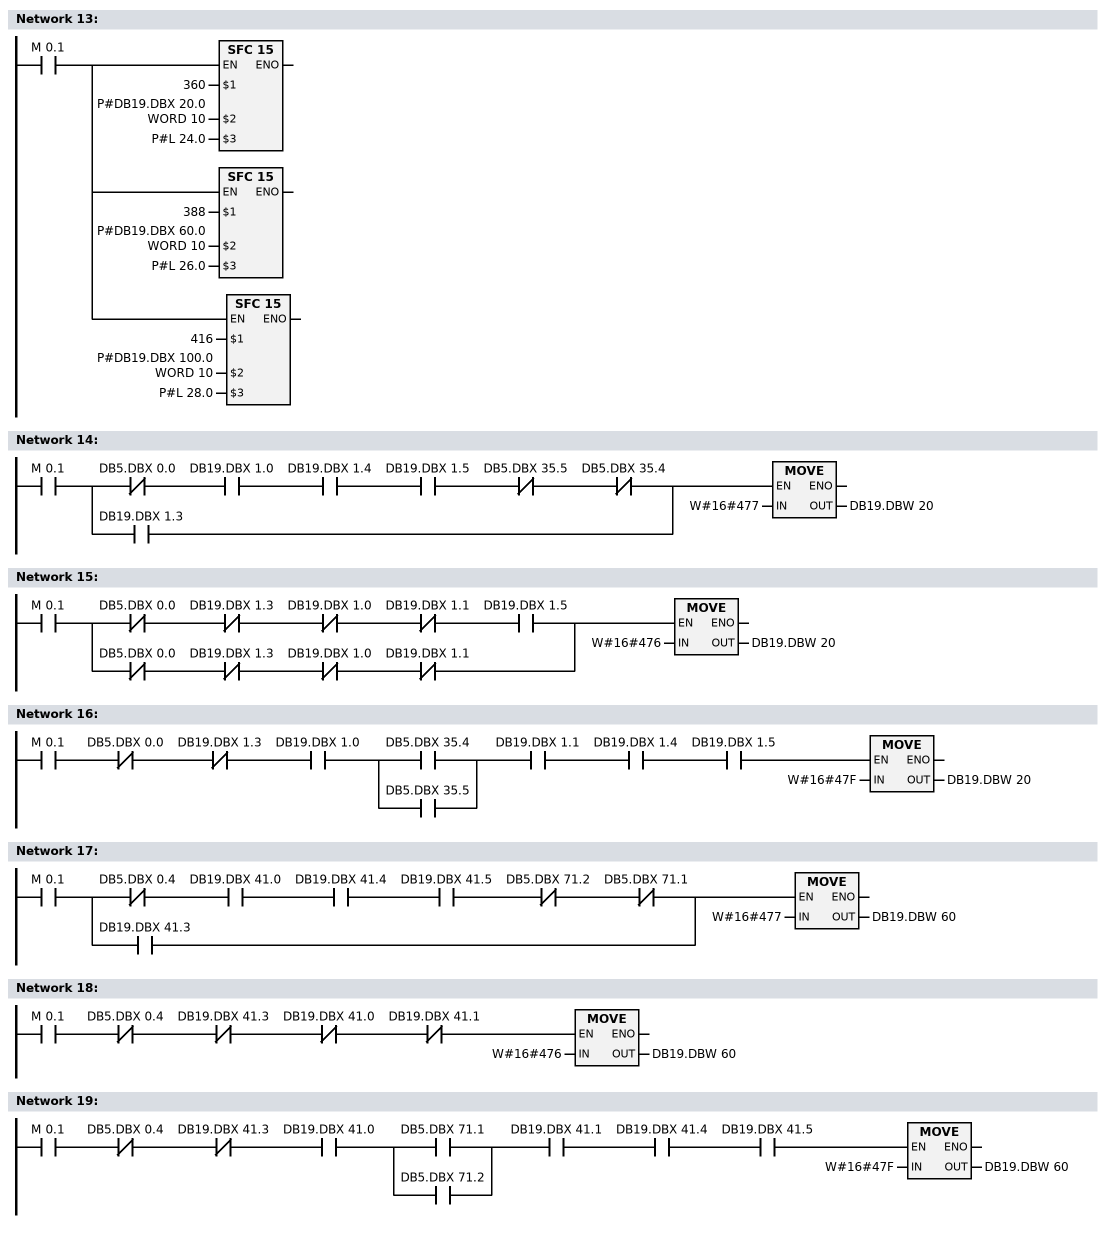
NETWORK
TITLE =
      A     M 0.1;
      =     L 36.0;
      A     L 36.0;
      JNB   M019;
      CALL  SFC 15 (
           $1                       := 360,
           $2                       := P#DB19.DBX 20.0 WORD 10,
           $3                       := P#L 24.0);
M019: NOP   0;
      A     L 36.0;
      JNB   M020;
      CALL  SFC 15 (
           $1                       := 388,
           $2                       := P#DB19.DBX 60.0 WORD 10,
           $3                       := P#L 26.0);
M020: NOP   0;
      A     L 36.0;
      JNB   M021;
      CALL  SFC 15 (
           $1                       := 416,
           $2                       := P#DB19.DBX 100.0 WORD 10,
           $3                       := P#L 28.0);
M021: NOP   0;
NETWORK
TITLE =
      A     M 0.1;
      A(;
      AN    DB5.DBX 0.0;
      A     DB19.DBX 1.0;
      A     DB19.DBX 1.4;
      A     DB19.DBX 1.5;
      AN    DB5.DBX 35.5;
      AN    DB5.DBX 35.4;
      O     DB19.DBX 1.3;
      );
      JNB   M022;
      L     W#16#477;
      T     DB19.DBW 20;
M022: NOP   0;
NETWORK
TITLE =
      A     M 0.1;
      A(;
      AN    DB5.DBX 0.0;
      AN    DB19.DBX 1.3;
      AN    DB19.DBX 1.0;
      AN    DB19.DBX 1.1;
      A     DB19.DBX 1.5;
      O;
      AN    DB5.DBX 0.0;
      AN    DB19.DBX 1.3;
      AN    DB19.DBX 1.0;
      AN    DB19.DBX 1.1;
      );
      JNB   M023;
      L     W#16#476;
      T     DB19.DBW 20;
M023: NOP   0;
NETWORK
TITLE =
      A     M 0.1;
      AN    DB5.DBX 0.0;
      AN    DB19.DBX 1.3;
      A     DB19.DBX 1.0;
      A(;
      O     DB5.DBX 35.4;
      O     DB5.DBX 35.5;
      );
      A     DB19.DBX 1.1;
      A     DB19.DBX 1.4;
      A     DB19.DBX 1.5;
      JNB   M024;
      L     W#16#47F;
      T     DB19.DBW 20;
M024: NOP   0;
NETWORK
TITLE =
      A     M 0.1;
      A(;
      AN    DB5.DBX 0.4;
      A     DB19.DBX 41.0;
      A     DB19.DBX 41.4;
      A     DB19.DBX 41.5;
      AN    DB5.DBX 71.2;
      AN    DB5.DBX 71.1;
      O     DB19.DBX 41.3;
      );
      JNB   M025;
      L     W#16#477;
      T     DB19.DBW 60;
M025: NOP   0;
NETWORK
TITLE =
      A     M 0.1;
      AN    DB5.DBX 0.4;
      AN    DB19.DBX 41.3;
      AN    DB19.DBX 41.0;
      AN    DB19.DBX 41.1;
      JNB   M026;
      L     W#16#476;
      T     DB19.DBW 60;
M026: NOP   0;
NETWORK
TITLE =
      A     M 0.1;
      AN    DB5.DBX 0.4;
      AN    DB19.DBX 41.3;
      A     DB19.DBX 41.0;
      A(;
      O     DB5.DBX 71.1;
      O     DB5.DBX 71.2;
      );
      A     DB19.DBX 41.1;
      A     DB19.DBX 41.4;
      A     DB19.DBX 41.5;
      JNB   M027;
      L     W#16#47F;
      T     DB19.DBW 60;
M027: NOP   0;
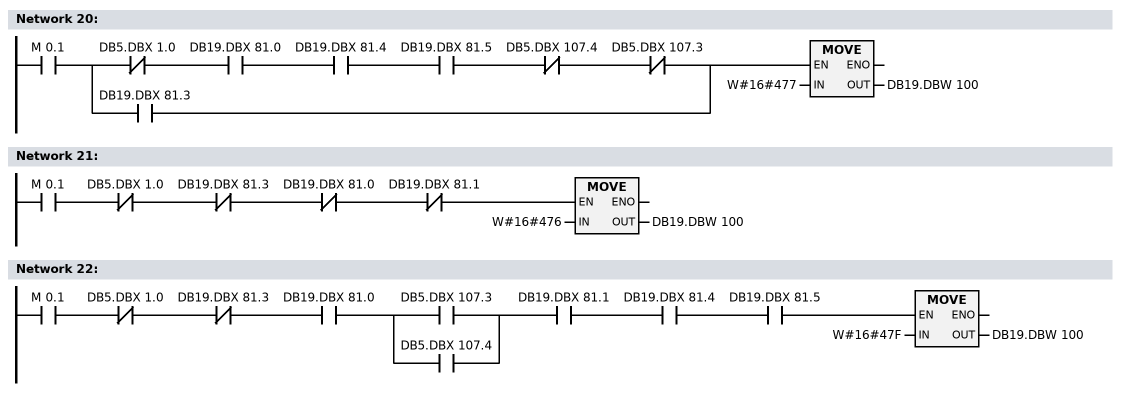
NETWORK
TITLE =
      A     M 0.1;
      A(;
      AN    DB5.DBX 1.0;
      A     DB19.DBX 81.0;
      A     DB19.DBX 81.4;
      A     DB19.DBX 81.5;
      AN    DB5.DBX 107.4;
      AN    DB5.DBX 107.3;
      O     DB19.DBX 81.3;
      );
      JNB   M028;
      L     W#16#477;
      T     DB19.DBW 100;
M028: NOP   0;
NETWORK
TITLE =
      A     M 0.1;
      AN    DB5.DBX 1.0;
      AN    DB19.DBX 81.3;
      AN    DB19.DBX 81.0;
      AN    DB19.DBX 81.1;
      JNB   M029;
      L     W#16#476;
      T     DB19.DBW 100;
M029: NOP   0;
NETWORK
TITLE =
      A     M 0.1;
      AN    DB5.DBX 1.0;
      AN    DB19.DBX 81.3;
      A     DB19.DBX 81.0;
      A(;
      O     DB5.DBX 107.3;
      O     DB5.DBX 107.4;
      );
      A     DB19.DBX 81.1;
      A     DB19.DBX 81.4;
      A     DB19.DBX 81.5;
      JNB   M030;
      L     W#16#47F;
      T     DB19.DBW 100;
M030: NOP   0;
END_FUNCTION

FUNCTION FC 13 : VOID
AUTHOR : Arun
VERSION : 0.1
BEGIN
// (block stored without names or comments; labels and parameter names are numbered)
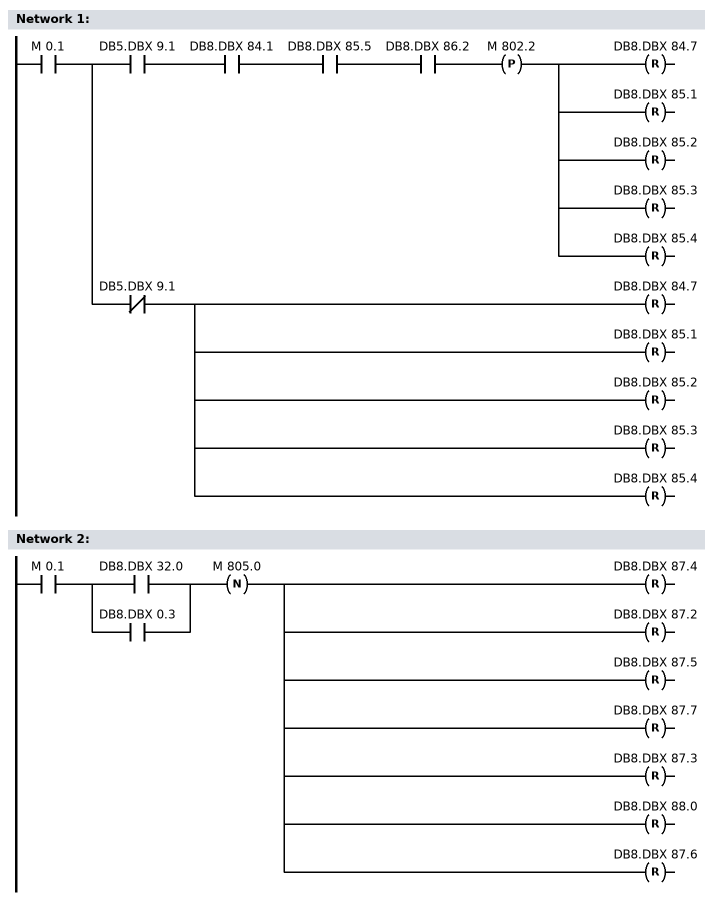
NETWORK
TITLE =
      A     M 0.1;
      =     L 0.0;
      A     L 0.0;
      A     DB5.DBX 9.1;
      A     DB8.DBX 84.1;
      A     DB8.DBX 85.5;
      A     DB8.DBX 86.2;
      FP    M 802.2;
      R     DB8.DBX 84.7;
      R     DB8.DBX 85.1;
      R     DB8.DBX 85.2;
      R     DB8.DBX 85.3;
      R     DB8.DBX 85.4;
      A     L 0.0;
      AN    DB5.DBX 9.1;
      R     DB8.DBX 84.7;
      R     DB8.DBX 85.1;
      R     DB8.DBX 85.2;
      R     DB8.DBX 85.3;
      R     DB8.DBX 85.4;
NETWORK
TITLE =
      A     M 0.1;
      A(;
      O     DB8.DBX 32.0;
      O     DB8.DBX 0.3;
      );
      FN    M 805.0;
      R     DB8.DBX 87.4;
      R     DB8.DBX 87.2;
      R     DB8.DBX 87.5;
      R     DB8.DBX 87.7;
      R     DB8.DBX 87.3;
      R     DB8.DBX 88.0;
      R     DB8.DBX 87.6;
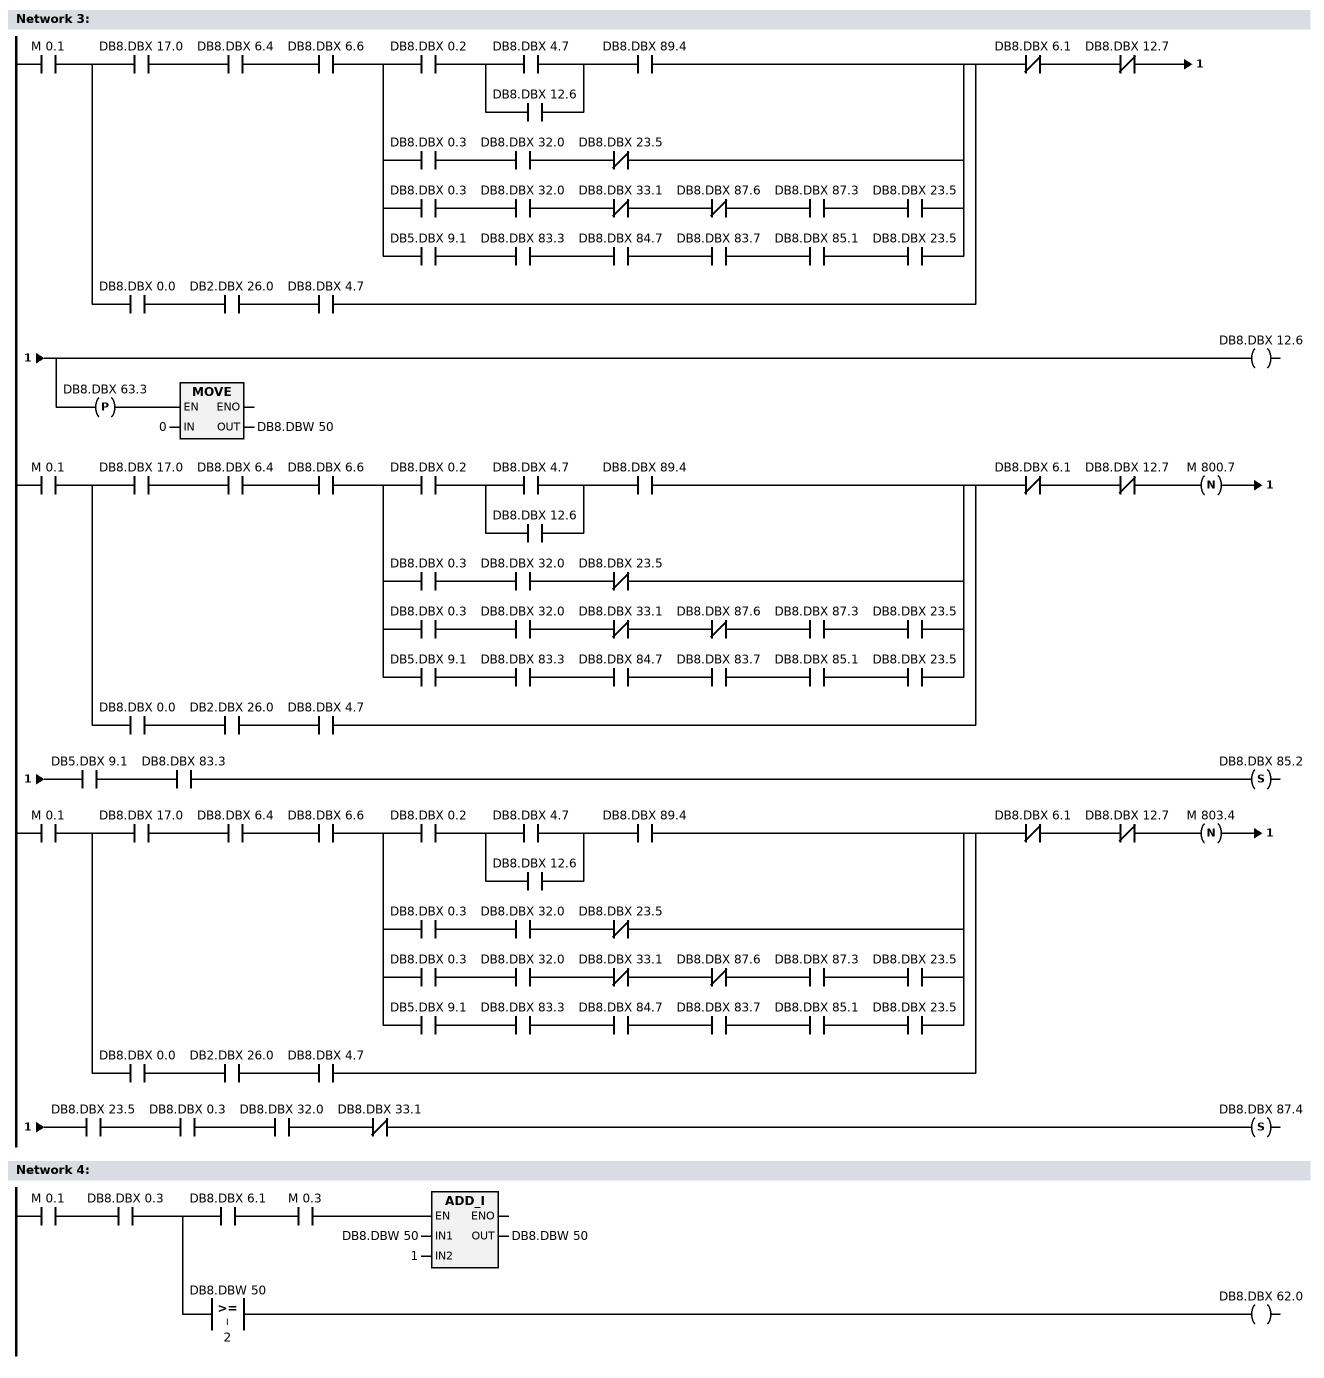
NETWORK
TITLE =
      A     M 0.1;
      A(;
      A     DB8.DBX 17.0;
      A     DB8.DBX 6.4;
      A     DB8.DBX 6.6;
      A(;
      A     DB8.DBX 0.2;
      A(;
      O     DB8.DBX 4.7;
      O     DB8.DBX 12.6;
      );
      A     DB8.DBX 89.4;
      O;
      A     DB8.DBX 0.3;
      A     DB8.DBX 32.0;
      AN    DB8.DBX 23.5;
      O;
      A     DB8.DBX 0.3;
      A     DB8.DBX 32.0;
      AN    DB8.DBX 33.1;
      AN    DB8.DBX 87.6;
      A     DB8.DBX 87.3;
      A     DB8.DBX 23.5;
      O;
      A     DB5.DBX 9.1;
      A     DB8.DBX 83.3;
      A     DB8.DBX 84.7;
      A     DB8.DBX 83.7;
      A     DB8.DBX 85.1;
      A     DB8.DBX 23.5;
      );
      O;
      A     DB8.DBX 0.0;
      A     DB2.DBX 26.0;
      A     DB8.DBX 4.7;
      );
      AN    DB8.DBX 6.1;
      AN    DB8.DBX 12.7;
      =     L 0.0;
      A     L 0.0;
      BLD   102;
      =     DB8.DBX 12.6;
      A     L 0.0;
      FP    DB8.DBX 63.3;
      JNB   M001;
      L     0;
      T     DB8.DBW 50;
M001: NOP   0;
      A(;
      A     L 0.0;
      FN    M 800.7;
      );
      A     DB5.DBX 9.1;
      A     DB8.DBX 83.3;
      S     DB8.DBX 85.2;
      A(;
      A     L 0.0;
      FN    M 803.4;
      );
      A     DB8.DBX 23.5;
      A     DB8.DBX 0.3;
      A     DB8.DBX 32.0;
      AN    DB8.DBX 33.1;
      S     DB8.DBX 87.4;
NETWORK
TITLE =
      A     M 0.1;
      A     DB8.DBX 0.3;
      =     L 0.0;
      A     L 0.0;
      A     DB8.DBX 6.1;
      A     M 0.3;
      JNB   M002;
      L     DB8.DBW 50;
      L     1;
      +I;
      T     DB8.DBW 50;
M002: NOP   0;
      A     L 0.0;
      A(;
      L     DB8.DBW 50;
      L     2;
      >=I;
      );
      =     DB8.DBX 62.0;
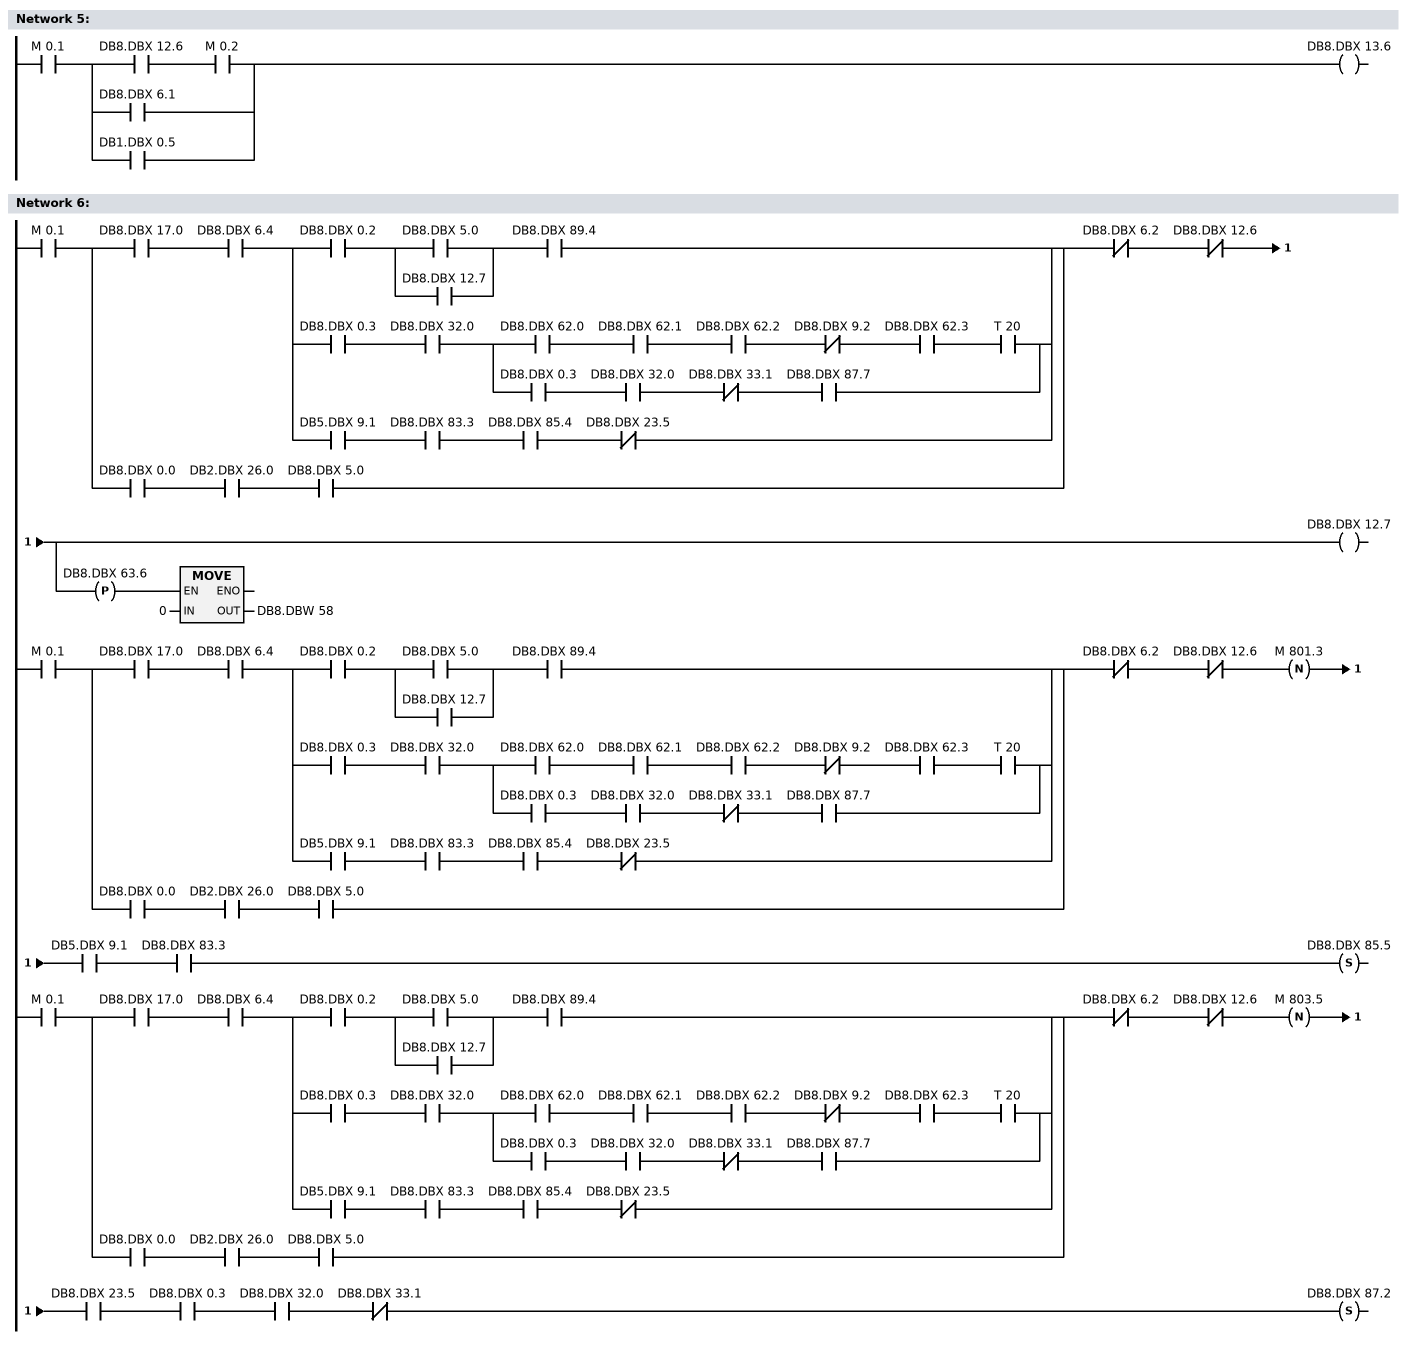
NETWORK
TITLE =
      A     M 0.1;
      A(;
      A     DB8.DBX 12.6;
      A     M 0.2;
      O     DB8.DBX 6.1;
      O     DB1.DBX 0.5;
      );
      =     DB8.DBX 13.6;
NETWORK
TITLE =
      A     M 0.1;
      A(;
      A     DB8.DBX 17.0;
      A     DB8.DBX 6.4;
      A(;
      A     DB8.DBX 0.2;
      A(;
      O     DB8.DBX 5.0;
      O     DB8.DBX 12.7;
      );
      A     DB8.DBX 89.4;
      O;
      A     DB8.DBX 0.3;
      A     DB8.DBX 32.0;
      A(;
      A     DB8.DBX 62.0;
      A     DB8.DBX 62.1;
      A     DB8.DBX 62.2;
      AN    DB8.DBX 9.2;
      A     DB8.DBX 62.3;
      A     T 20;
      O;
      A     DB8.DBX 0.3;
      A     DB8.DBX 32.0;
      AN    DB8.DBX 33.1;
      A     DB8.DBX 87.7;
      );
      O;
      A     DB5.DBX 9.1;
      A     DB8.DBX 83.3;
      A     DB8.DBX 85.4;
      AN    DB8.DBX 23.5;
      );
      O;
      A     DB8.DBX 0.0;
      A     DB2.DBX 26.0;
      A     DB8.DBX 5.0;
      );
      AN    DB8.DBX 6.2;
      AN    DB8.DBX 12.6;
      =     L 0.0;
      A     L 0.0;
      BLD   102;
      =     DB8.DBX 12.7;
      A     L 0.0;
      FP    DB8.DBX 63.6;
      JNB   M003;
      L     0;
      T     DB8.DBW 58;
M003: NOP   0;
      A(;
      A     L 0.0;
      FN    M 801.3;
      );
      A     DB5.DBX 9.1;
      A     DB8.DBX 83.3;
      S     DB8.DBX 85.5;
      A(;
      A     L 0.0;
      FN    M 803.5;
      );
      A     DB8.DBX 23.5;
      A     DB8.DBX 0.3;
      A     DB8.DBX 32.0;
      AN    DB8.DBX 33.1;
      S     DB8.DBX 87.2;
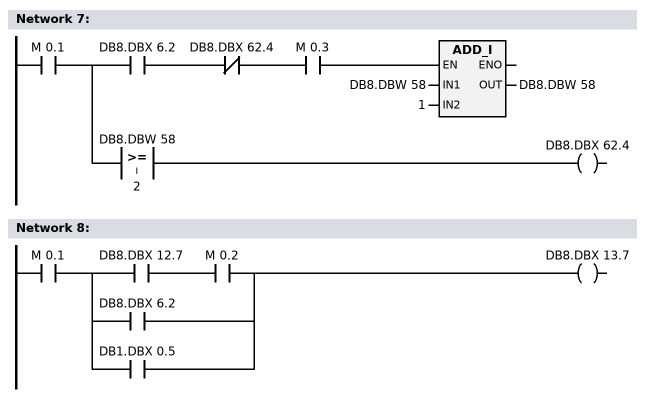
NETWORK
TITLE =
      A     M 0.1;
      =     L 0.0;
      A     L 0.0;
      A     DB8.DBX 6.2;
      AN    DB8.DBX 62.4;
      A     M 0.3;
      JNB   M004;
      L     DB8.DBW 58;
      L     1;
      +I;
      T     DB8.DBW 58;
M004: NOP   0;
      A     L 0.0;
      A(;
      L     DB8.DBW 58;
      L     2;
      >=I;
      );
      =     DB8.DBX 62.4;
NETWORK
TITLE =
      A     M 0.1;
      A(;
      A     DB8.DBX 12.7;
      A     M 0.2;
      O     DB8.DBX 6.2;
      O     DB1.DBX 0.5;
      );
      =     DB8.DBX 13.7;
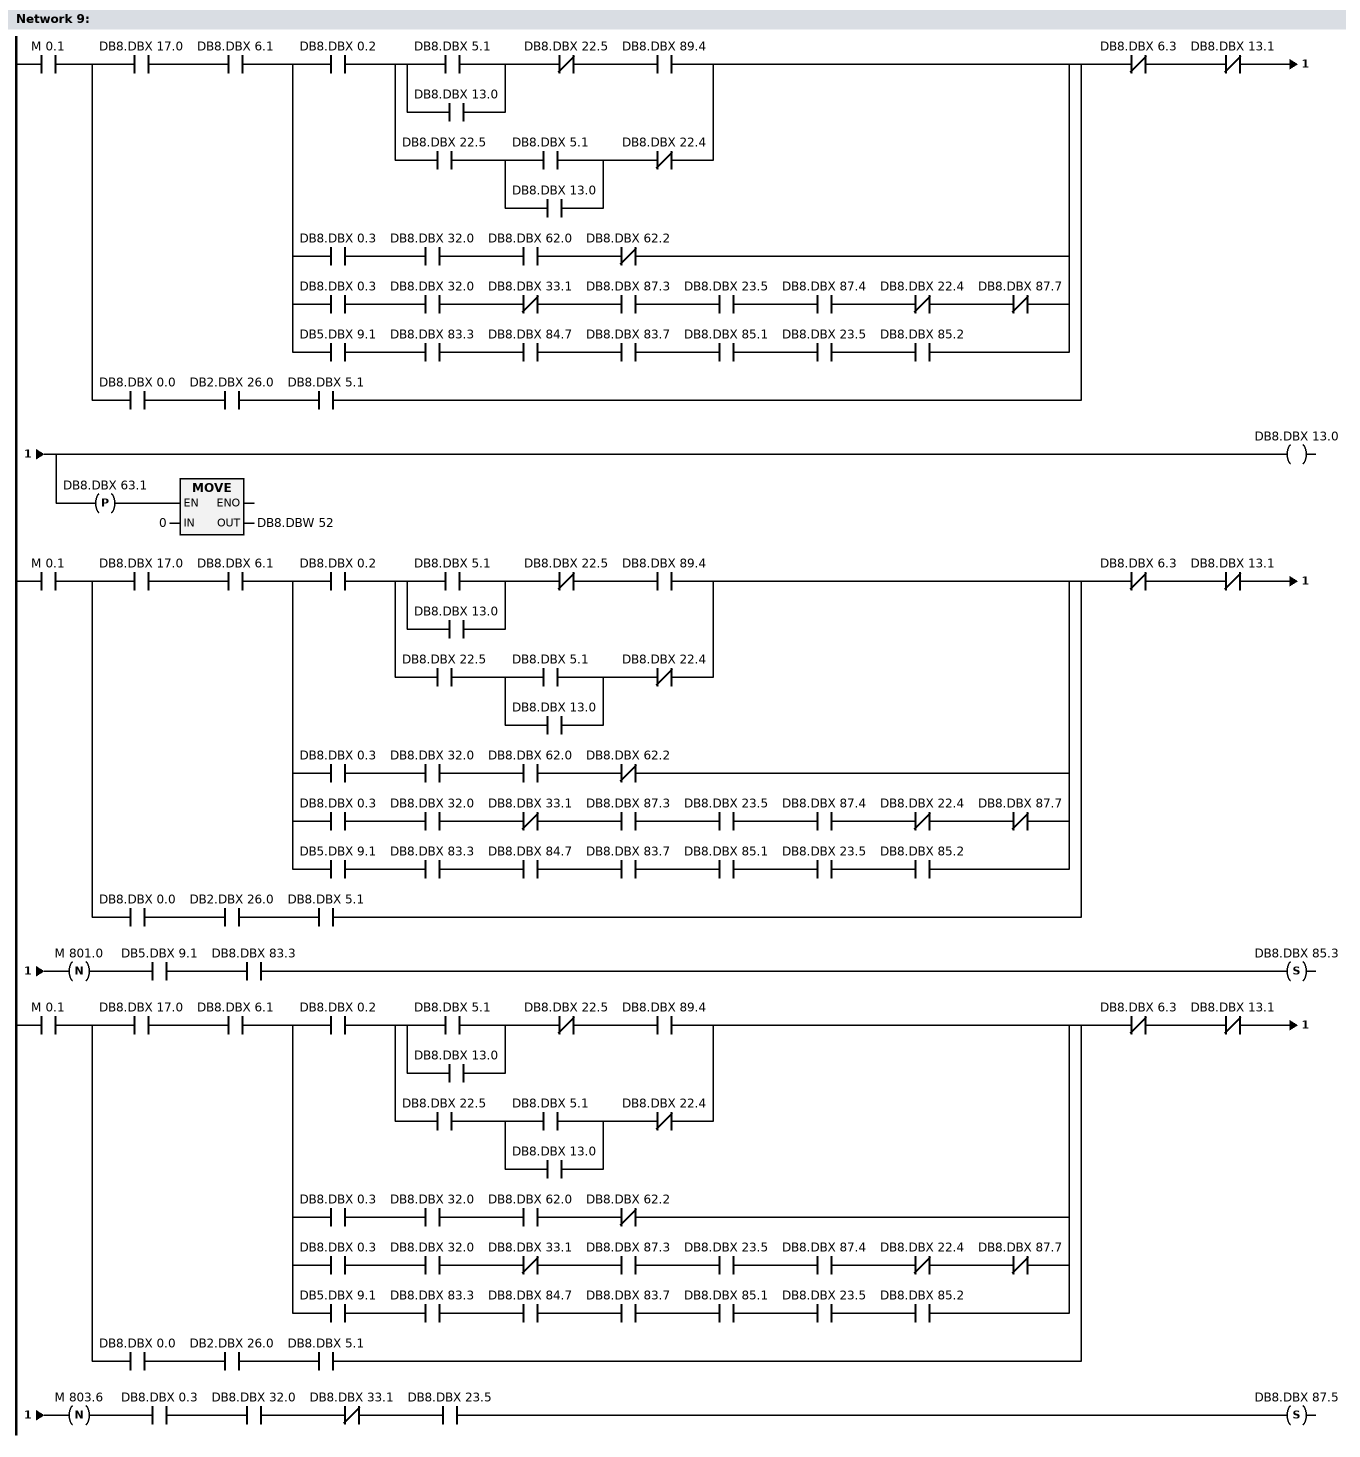
NETWORK
TITLE =
      A     M 0.1;
      A(;
      A     DB8.DBX 17.0;
      A     DB8.DBX 6.1;
      A(;
      A     DB8.DBX 0.2;
      A(;
      A(;
      O     DB8.DBX 5.1;
      O     DB8.DBX 13.0;
      );
      AN    DB8.DBX 22.5;
      A     DB8.DBX 89.4;
      O;
      A     DB8.DBX 22.5;
      A(;
      O     DB8.DBX 5.1;
      O     DB8.DBX 13.0;
      );
      AN    DB8.DBX 22.4;
      );
      O;
      A     DB8.DBX 0.3;
      A     DB8.DBX 32.0;
      A     DB8.DBX 62.0;
      AN    DB8.DBX 62.2;
      O;
      A     DB8.DBX 0.3;
      A     DB8.DBX 32.0;
      AN    DB8.DBX 33.1;
      A     DB8.DBX 87.3;
      A     DB8.DBX 23.5;
      A     DB8.DBX 87.4;
      AN    DB8.DBX 22.4;
      AN    DB8.DBX 87.7;
      O;
      A     DB5.DBX 9.1;
      A     DB8.DBX 83.3;
      A     DB8.DBX 84.7;
      A     DB8.DBX 83.7;
      A     DB8.DBX 85.1;
      A     DB8.DBX 23.5;
      A     DB8.DBX 85.2;
      );
      O;
      A     DB8.DBX 0.0;
      A     DB2.DBX 26.0;
      A     DB8.DBX 5.1;
      );
      AN    DB8.DBX 6.3;
      AN    DB8.DBX 13.1;
      =     L 0.0;
      A     L 0.0;
      BLD   102;
      =     DB8.DBX 13.0;
      A     L 0.0;
      FP    DB8.DBX 63.1;
      JNB   M005;
      L     0;
      T     DB8.DBW 52;
M005: NOP   0;
      A(;
      A     L 0.0;
      FN    M 801.0;
      );
      A     DB5.DBX 9.1;
      A     DB8.DBX 83.3;
      S     DB8.DBX 85.3;
      A(;
      A     L 0.0;
      FN    M 803.6;
      );
      A     DB8.DBX 0.3;
      A     DB8.DBX 32.0;
      AN    DB8.DBX 33.1;
      A     DB8.DBX 23.5;
      S     DB8.DBX 87.5;
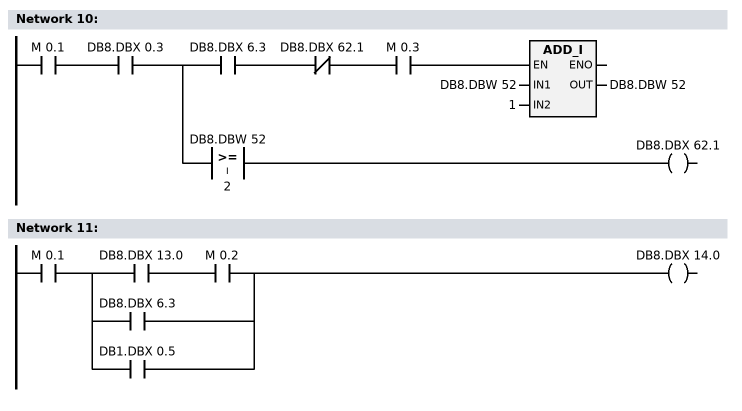
NETWORK
TITLE =
      A     M 0.1;
      A     DB8.DBX 0.3;
      =     L 0.0;
      A     L 0.0;
      A     DB8.DBX 6.3;
      AN    DB8.DBX 62.1;
      A     M 0.3;
      JNB   M006;
      L     DB8.DBW 52;
      L     1;
      +I;
      T     DB8.DBW 52;
M006: NOP   0;
      A     L 0.0;
      A(;
      L     DB8.DBW 52;
      L     2;
      >=I;
      );
      =     DB8.DBX 62.1;
NETWORK
TITLE =
      A     M 0.1;
      A(;
      A     DB8.DBX 13.0;
      A     M 0.2;
      O     DB8.DBX 6.3;
      O     DB1.DBX 0.5;
      );
      =     DB8.DBX 14.0;
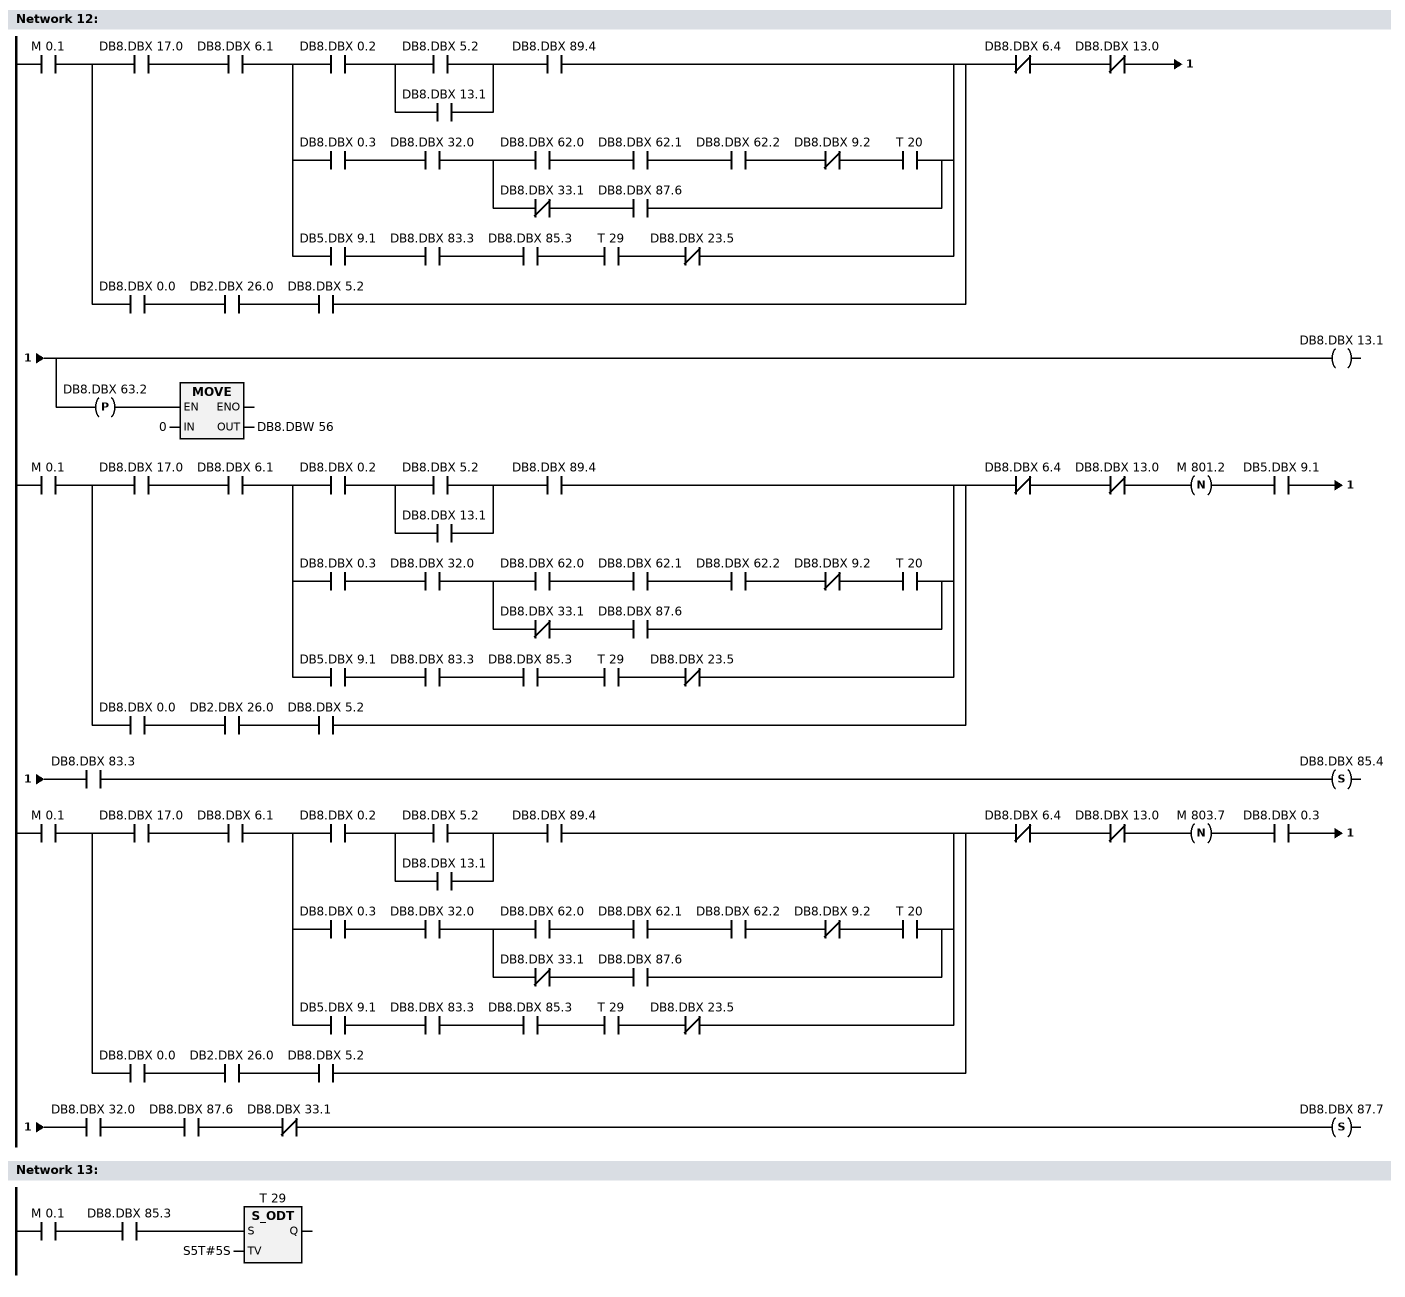
NETWORK
TITLE =
      A     M 0.1;
      A(;
      A     DB8.DBX 17.0;
      A     DB8.DBX 6.1;
      A(;
      A     DB8.DBX 0.2;
      A(;
      O     DB8.DBX 5.2;
      O     DB8.DBX 13.1;
      );
      A     DB8.DBX 89.4;
      O;
      A     DB8.DBX 0.3;
      A     DB8.DBX 32.0;
      A(;
      A     DB8.DBX 62.0;
      A     DB8.DBX 62.1;
      A     DB8.DBX 62.2;
      AN    DB8.DBX 9.2;
      A     T 20;
      O;
      AN    DB8.DBX 33.1;
      A     DB8.DBX 87.6;
      );
      O;
      A     DB5.DBX 9.1;
      A     DB8.DBX 83.3;
      A     DB8.DBX 85.3;
      A     T 29;
      AN    DB8.DBX 23.5;
      );
      O;
      A     DB8.DBX 0.0;
      A     DB2.DBX 26.0;
      A     DB8.DBX 5.2;
      );
      AN    DB8.DBX 6.4;
      AN    DB8.DBX 13.0;
      =     L 0.0;
      A     L 0.0;
      BLD   102;
      =     DB8.DBX 13.1;
      A     L 0.0;
      FP    DB8.DBX 63.2;
      JNB   M007;
      L     0;
      T     DB8.DBW 56;
M007: NOP   0;
      A(;
      A     L 0.0;
      FN    M 801.2;
      );
      A     DB5.DBX 9.1;
      A     DB8.DBX 83.3;
      S     DB8.DBX 85.4;
      A(;
      A     L 0.0;
      FN    M 803.7;
      );
      A     DB8.DBX 0.3;
      A     DB8.DBX 32.0;
      A     DB8.DBX 87.6;
      AN    DB8.DBX 33.1;
      S     DB8.DBX 87.7;
NETWORK
TITLE =
      A     M 0.1;
      A     DB8.DBX 85.3;
      L     S5T#5S;
      SD    T 29;
      NOP   0;
      NOP   0;
      NOP   0;
      NOP   0;
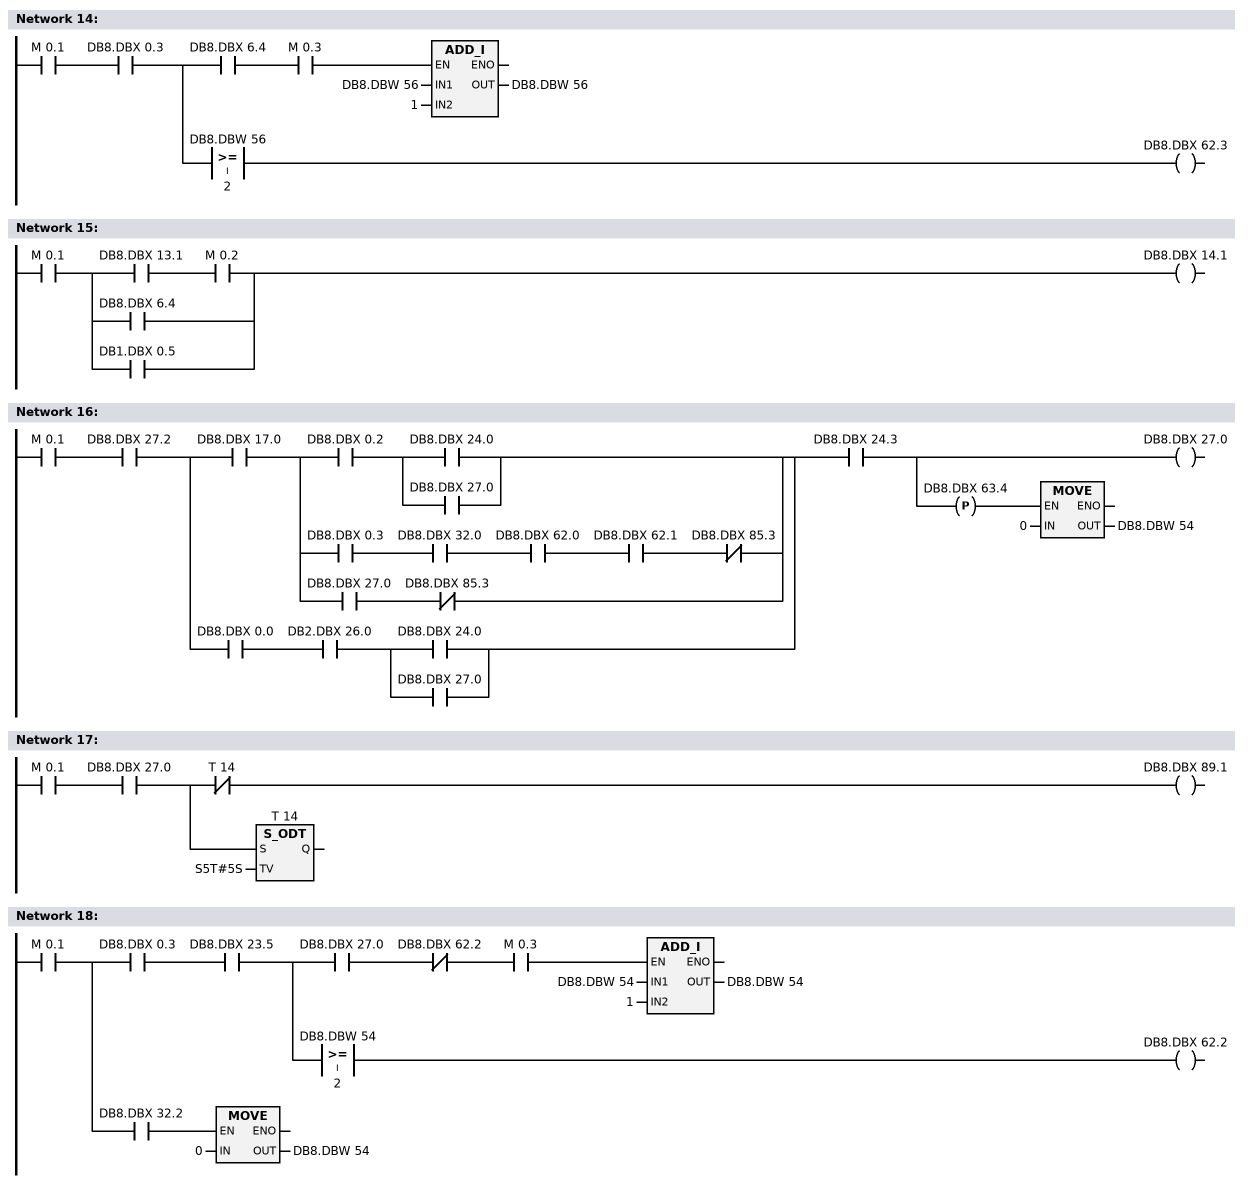
NETWORK
TITLE =
      A     M 0.1;
      A     DB8.DBX 0.3;
      =     L 0.0;
      A     L 0.0;
      A     DB8.DBX 6.4;
      A     M 0.3;
      JNB   M008;
      L     DB8.DBW 56;
      L     1;
      +I;
      T     DB8.DBW 56;
M008: NOP   0;
      A     L 0.0;
      A(;
      L     DB8.DBW 56;
      L     2;
      >=I;
      );
      =     DB8.DBX 62.3;
NETWORK
TITLE =
      A     M 0.1;
      A(;
      A     DB8.DBX 13.1;
      A     M 0.2;
      O     DB8.DBX 6.4;
      O     DB1.DBX 0.5;
      );
      =     DB8.DBX 14.1;
NETWORK
TITLE =
      A     M 0.1;
      A     DB8.DBX 27.2;
      A(;
      A     DB8.DBX 17.0;
      A(;
      A     DB8.DBX 0.2;
      A(;
      O     DB8.DBX 24.0;
      O     DB8.DBX 27.0;
      );
      O;
      A     DB8.DBX 0.3;
      A     DB8.DBX 32.0;
      A     DB8.DBX 62.0;
      A     DB8.DBX 62.1;
      AN    DB8.DBX 85.3;
      O;
      A     DB8.DBX 27.0;
      AN    DB8.DBX 85.3;
      );
      O;
      A     DB8.DBX 0.0;
      A     DB2.DBX 26.0;
      A(;
      O     DB8.DBX 24.0;
      O     DB8.DBX 27.0;
      );
      );
      A     DB8.DBX 24.3;
      =     L 0.0;
      A     L 0.0;
      BLD   102;
      =     DB8.DBX 27.0;
      A     L 0.0;
      FP    DB8.DBX 63.4;
      JNB   M009;
      L     0;
      T     DB8.DBW 54;
M009: NOP   0;
NETWORK
TITLE =
      A     M 0.1;
      A     DB8.DBX 27.0;
      =     L 0.0;
      A     L 0.0;
      AN    T 14;
      =     DB8.DBX 89.1;
      A     L 0.0;
      L     S5T#5S;
      SD    T 14;
      NOP   0;
      NOP   0;
      NOP   0;
      NOP   0;
NETWORK
TITLE =
      A     M 0.1;
      =     L 0.0;
      A     L 0.0;
      A     DB8.DBX 0.3;
      A     DB8.DBX 23.5;
      =     L 0.1;
      A     L 0.1;
      A     DB8.DBX 27.0;
      AN    DB8.DBX 62.2;
      A     M 0.3;
      JNB   M010;
      L     DB8.DBW 54;
      L     1;
      +I;
      T     DB8.DBW 54;
M010: NOP   0;
      A     L 0.1;
      A(;
      L     DB8.DBW 54;
      L     2;
      >=I;
      );
      =     DB8.DBX 62.2;
      A     L 0.0;
      A     DB8.DBX 32.2;
      JNB   M011;
      L     0;
      T     DB8.DBW 54;
M011: NOP   0;
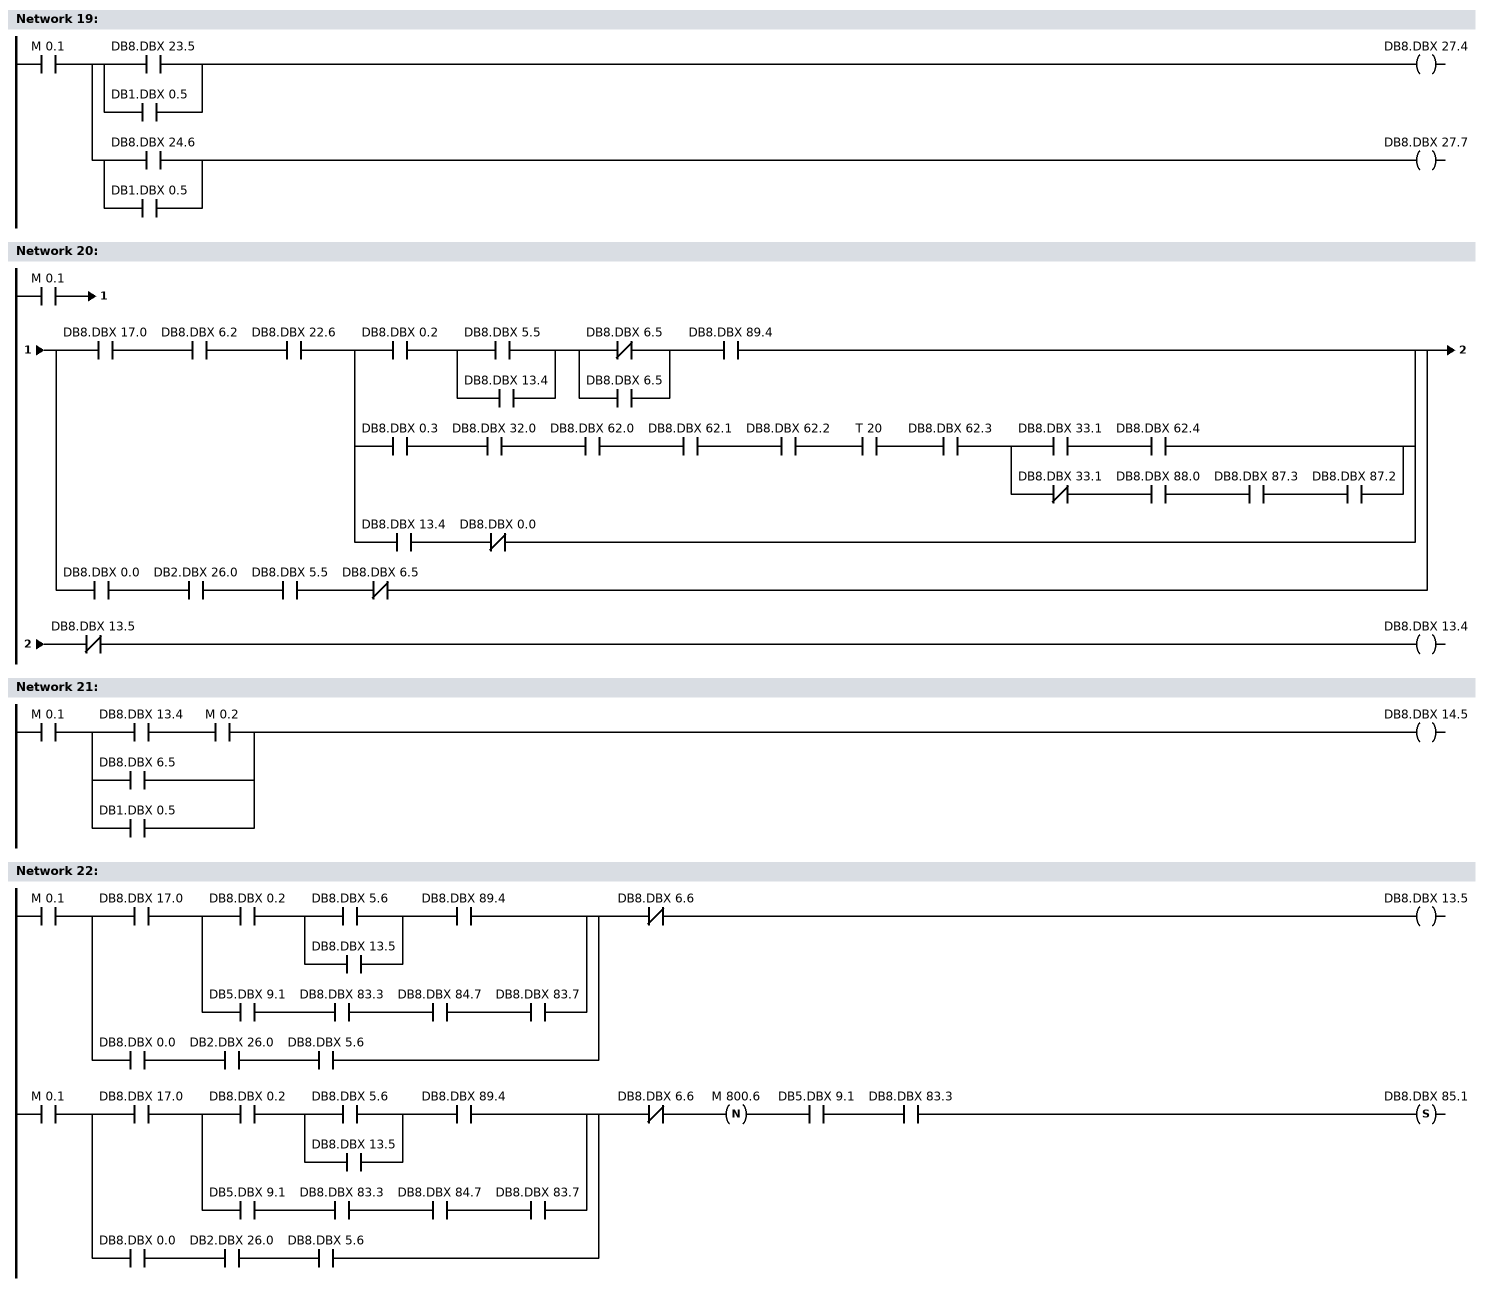
NETWORK
TITLE =
      A     M 0.1;
      =     L 0.0;
      A     L 0.0;
      A(;
      O     DB8.DBX 23.5;
      O     DB1.DBX 0.5;
      );
      =     DB8.DBX 27.4;
      A     L 0.0;
      A(;
      O     DB8.DBX 24.6;
      O     DB1.DBX 0.5;
      );
      =     DB8.DBX 27.7;
NETWORK
TITLE =
      A     M 0.1;
      A(;
      A     DB8.DBX 17.0;
      A     DB8.DBX 6.2;
      A     DB8.DBX 22.6;
      A(;
      A     DB8.DBX 0.2;
      A(;
      O     DB8.DBX 5.5;
      O     DB8.DBX 13.4;
      );
      A(;
      ON    DB8.DBX 6.5;
      O     DB8.DBX 6.5;
      );
      A     DB8.DBX 89.4;
      O;
      A     DB8.DBX 0.3;
      A     DB8.DBX 32.0;
      A     DB8.DBX 62.0;
      A     DB8.DBX 62.1;
      A     DB8.DBX 62.2;
      A     T 20;
      A     DB8.DBX 62.3;
      A(;
      A     DB8.DBX 33.1;
      A     DB8.DBX 62.4;
      O;
      AN    DB8.DBX 33.1;
      A     DB8.DBX 88.0;
      A     DB8.DBX 87.3;
      A     DB8.DBX 87.2;
      );
      O;
      A     DB8.DBX 13.4;
      AN    DB8.DBX 0.0;
      );
      O;
      A     DB8.DBX 0.0;
      A     DB2.DBX 26.0;
      A     DB8.DBX 5.5;
      AN    DB8.DBX 6.5;
      );
      AN    DB8.DBX 13.5;
      =     DB8.DBX 13.4;
NETWORK
TITLE =
      A     M 0.1;
      A(;
      A     DB8.DBX 13.4;
      A     M 0.2;
      O     DB8.DBX 6.5;
      O     DB1.DBX 0.5;
      );
      =     DB8.DBX 14.5;
NETWORK
TITLE =
      A     M 0.1;
      A(;
      A     DB8.DBX 17.0;
      A(;
      A     DB8.DBX 0.2;
      A(;
      O     DB8.DBX 5.6;
      O     DB8.DBX 13.5;
      );
      A     DB8.DBX 89.4;
      O;
      A     DB5.DBX 9.1;
      A     DB8.DBX 83.3;
      A     DB8.DBX 84.7;
      A     DB8.DBX 83.7;
      );
      O;
      A     DB8.DBX 0.0;
      A     DB2.DBX 26.0;
      A     DB8.DBX 5.6;
      );
      AN    DB8.DBX 6.6;
      =     L 0.0;
      A     L 0.0;
      BLD   102;
      =     DB8.DBX 13.5;
      A(;
      A     L 0.0;
      FN    M 800.6;
      );
      A     DB5.DBX 9.1;
      A     DB8.DBX 83.3;
      S     DB8.DBX 85.1;
